	//--- delete and shift 
		IF udiNbOfCarrier >= 1 THEN
			//--- Check if Carrier is outside
				//--- zero is not inside start and end pos 
			FOR udiTraceArrayIndex := 1 TO c_udiTraceObjects DO
				IF audiTraceCarrierIndex[udiTraceArrayIndex] = 0 THEN
					CONTINUE;
				END_IF
				IF i_lrStartPos < i_lrEndPos THEN 
					IF fbMulticarrier.raifCarrier[audiTraceCarrierIndex[udiTraceArrayIndex]].ifFeedback.ifFeedbackMotionValues.lrRefTrackPosition > i_lrEndPos
						OR fbMulticarrier.raifCarrier[audiTraceCarrierIndex[udiTraceArrayIndex]].ifFeedback.ifFeedbackMotionValues.lrRefTrackPosition < i_lrStartPos
					THEN
						xCarrierIsOutside := TRUE;
						EXIT;
					END_IF
					
				//--- zero is inside start and end pos  
				ELSIF i_lrStartPos > i_lrEndPos THEN 
					IF fbMulticarrier.raifCarrier[audiTraceCarrierIndex[udiTraceArrayIndex]].ifFeedback.ifFeedbackMotionValues.lrRefTrackPosition > i_lrEndPos
						AND fbMulticarrier.raifCarrier[audiTraceCarrierIndex[udiTraceArrayIndex]].ifFeedback.ifFeedbackMotionValues.lrRefTrackPosition < i_lrStartPos
					THEN
						xCarrierIsOutside := TRUE;
						EXIT;
					END_IF
				END_IF
			END_FOR
			
			IF xCarrierIsOutside THEN
				xCarrierIsOutside := FALSE;
				udiNbOfCarrier := udiNbOfCarrier -1;
				axCarrierArrayIsBlocked[udiTraceArrayIndex] := FALSE;
				audiTraceCarrierIndex[udiTraceArrayIndex] := 0;
			END_IF
		END_IF
END_METHOD

ACTION ExceptionControl_Action:
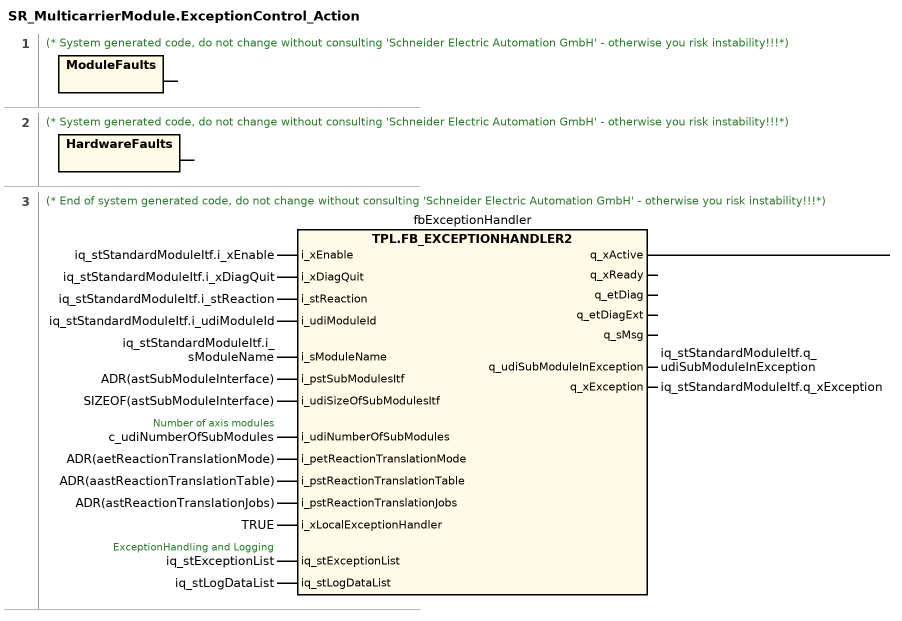
// NETWORK 1
// (* System generated code, do not change without consulting 'Schneider Electric Automation GmbH' - otherwise you risk instability!!!*)
ModuleFaults();

// NETWORK 2
// (* System generated code, do not change without consulting 'Schneider Electric Automation GmbH' - otherwise you risk instability!!!*)
HardwareFaults();

// NETWORK 3
// (* End of system generated code, do not change without consulting 'Schneider Electric Automation GmbH' - otherwise you risk instability!!!*)
//   fbExceptionHandler: ExceptionHandling related variables
//   c_udiNumberOfSubModules: Number of axis modules
//   iq_stExceptionList: ExceptionHandling and Logging
fbExceptionHandler(
    i_xEnable := iq_stStandardModuleItf.i_xEnable,
    i_xDiagQuit := iq_stStandardModuleItf.i_xDiagQuit,
    i_stReaction := iq_stStandardModuleItf.i_stReaction,
    i_udiModuleId := iq_stStandardModuleItf.i_udiModuleId,
    i_sModuleName := iq_stStandardModuleItf.i_sModuleName,
    i_pstSubModulesItf := ADR(astSubModuleInterface),
    i_udiSizeOfSubModulesItf := SIZEOF(astSubModuleInterface),
    i_udiNumberOfSubModules := c_udiNumberOfSubModules,
    i_petReactionTranslationMode := ADR(aetReactionTranslationMode),
    i_pstReactionTranslationTable := ADR(aastReactionTranslationTable),
    i_pstReactionTranslationJobs := ADR(astReactionTranslationJobs),
    i_xLocalExceptionHandler := TRUE,
    iq_stExceptionList := iq_stExceptionList,
    iq_stLogDataList := iq_stLogDataList,
    q_udiSubModuleInException => iq_stStandardModuleItf.q_udiSubModuleInException,
    q_xException => iq_stStandardModuleItf.q_xException); // TPL.FB_EXCEPTIONHANDLER2
END_ACTION

ACTION HardwareFaults:
(* System generated code, do not change without consulting 'Schneider Electric Automation GmbH' - otherwise you risk instability!!! *)
// 
IF SystemConfiguration.G_ifController <> 0 THEN
	diDiagCode := SystemConfiguration.G_ifController.DiagCode; 
	IF diDiagCode <> diDiagCode_old THEN
		diDiagCode_old	:= diDiagCode;
		stDiagSource	:= SystemConfiguration.G_ifController.DiagSource;
		IF 			stDiagSource.udiType = SystemInterface.LXMMCS_TYPE.udiType 
			OR_ELSE stDiagSource.udiType =  SystemInterface.LXMMCC_TYPE.udiType 
		THEN 
			diDiagClass		:= SystemConfiguration.G_ifController.DiagClass;
			sDiagMsg		:= SystemConfiguration.G_ifController.DiagMsg;
			sInstanceName	:= 'UnknownDevice';
			SystemInterface.FC_GetObjNameByLogAddr(i_stLogAdr := stDiagSource, i_diMaxSize := SIZEOF(sInstanceName), iq_sName := sInstanceName);
			sDiagMsgExt := '';
			xSuccess := __QUERYINTERFACE(SystemConfiguration.G_ifController, ifDiagnosis);
			IF xSuccess AND (ifDiagnosis <> 0) THEN
				sDiagMsgExt := ifDiagnosis.DiagExtMsg;
			END_IF

			diDiagClass := SystemConfiguration.G_ifController.DiagClass;
			IF diDiagClass = 4 THEN
				stHardwareException.stReaction.axReaction[TPL.ET_Reaction.AsyncStop]  := TRUE;
				stHardwareException.stReaction.axReaction[TPL.ET_Reaction.SyncStopEL] := FALSE;
				stHardwareException.stReaction.axReaction[TPL.ET_Reaction.SyncStopEH] := FALSE;
			ELSIF diDiagClass = 3 THEN
				stHardwareException.stReaction.axReaction[TPL.ET_Reaction.AsyncStop]  := FALSE;
				stHardwareException.stReaction.axReaction[TPL.ET_Reaction.SyncStopEL] := TRUE;
				stHardwareException.stReaction.axReaction[TPL.ET_Reaction.SyncStopEH] := FALSE;
			ELSIF (diDiagClass = 2 OR diDiagClass = 1) THEN
				stHardwareException.stReaction.axReaction[TPL.ET_Reaction.AsyncStop]  := FALSE;
				stHardwareException.stReaction.axReaction[TPL.ET_Reaction.SyncStopEL] := FALSE;
				stHardwareException.stReaction.axReaction[TPL.ET_Reaction.SyncStopEH] := TRUE;
			END_IF
			
			stHardwareException.etDiag		:= GD.ET_Diag.DiagActive;
			stHardwareException.udiDiagExt	:= ET_DiagExt.SystemFatalException;								
			stHardwareException.sDiagExt	:= FC_EtDiagExtToString(stHardwareException.udiDiagExt);	
			stHardwareException.sMsg		:= PDL.FC_MultiConcat(	i_sString1 := STANDARD.CONCAT(sInstanceName, ' '),
																	i_sString2 := STANDARD.CONCAT(DINT_TO_STRING(diDiagCode), ' '), 
																	i_sString3 := STANDARD.CONCAT(sDiagMsg, ' '), 
																	i_sString4 := sDiagMsgExt);
																	
			stHardwareException.udiExceptionNumber := TPL.FC_GenerateExceptionNumber( i_etSource := TPL.ET_ExceptionSource.System, i_udiDiagExt := DINT_TO_UDINT(diDiagCode) );
			fbExceptionHandler.SetException(i_xExceptionActive	:= TRUE,
											iq_stException		:= stHardwareException,
											iq_stExceptionList	:= iq_stExceptionList);
		END_IF
	END_IF
END_IF
// (* End of system generated code, do not change without consulting 'Schneider Electric Automation GmbH' - otherwise you risk instability!!! *)
END_ACTION

ACTION Init_Exceptions:
(* System generated code, could be modified for your application *)
stUpdateStructsException.etDiag												:= GD.ET_Diag.UnexpectedProgramBehavior;
stUpdateStructsException.udiDiagExt											:= ET_DiagExt.UpdateStructsException;
stUpdateStructsException.sDiagExt											:= FC_EtDiagExtToString(stUpdateStructsException.udiDiagExt);
stUpdateStructsException.sMsg												:= '';	(* Replaced on usage *)
stUpdateStructsException.udiModuleId										:= iq_stStandardModuleItf.i_udiModuleId;
stUpdateStructsException.sModuleName										:= iq_stStandardModuleItf.i_sModuleName;
stUpdateStructsException.stReaction.axReaction[TPL.ET_Reaction.AsyncStop]	:= TRUE;
stUpdateStructsException.etSource											:= TPL.ET_ExceptionSource.NodeModule;
stUpdateStructsException.timDelayTime										:= T#0MS;
stUpdateStructsException.wHmiAttributes										:= 0;
stUpdateStructsException.xAutoQuit											:= FALSE;

stInitReactionsException.etDiag												:= GD.ET_Diag.UnexpectedProgramBehavior;
stInitReactionsException.udiDiagExt											:= ET_DiagExt.InitReactionsException;
stInitReactionsException.sDiagExt											:= FC_EtDiagExtToString(stInitReactionsException.udiDiagExt);
stInitReactionsException.sMsg												:= '';	(* Replaced on usage *)
stInitReactionsException.udiModuleId										:= iq_stStandardModuleItf.i_udiModuleId;
stInitReactionsException.sModuleName										:= iq_stStandardModuleItf.i_sModuleName;
stInitReactionsException.stReaction.axReaction[TPL.ET_Reaction.AsyncStop]	:= TRUE;
stInitReactionsException.etSource											:= TPL.ET_ExceptionSource.NodeModule;
stInitReactionsException.timDelayTime										:= T#0MS;
stInitReactionsException.wHmiAttributes										:= 0;
stInitReactionsException.xAutoQuit											:= FALSE;

stInitSubModulesException.etDiag											:= GD.ET_Diag.UnexpectedProgramBehavior;
stInitSubModulesException.udiDiagExt										:= ET_DiagExt.InitSubModulesException;
stInitSubModulesException.sDiagExt											:= FC_EtDiagExtToString(stInitSubModulesException.udiDiagExt);
stInitSubModulesException.sMsg												:= '';	(* Replaced on usage *)
stInitSubModulesException.udiModuleId										:= iq_stStandardModuleItf.i_udiModuleId;
stInitSubModulesException.sModuleName										:= iq_stStandardModuleItf.i_sModuleName;
stInitSubModulesException.stReaction.axReaction[TPL.ET_Reaction.AsyncStop]	:= TRUE;
stInitSubModulesException.etSource											:= TPL.ET_ExceptionSource.NodeModule;
stInitSubModulesException.timDelayTime										:= T#0MS;
stInitSubModulesException.wHmiAttributes									:= 0;
stInitSubModulesException.xAutoQuit											:= FALSE;

(*------------------------------------------------------------------------------------------*)
(* Init User Exceptions *)

	// TPL.ET_Reaction.AsyncStop
	// TPL.ET_Reaction.SyncStopEL
	// TPL.ET_Reaction.SyncStopEH
	// TPL.ET_Reaction.StopEndOfCycle
	// TPL.ET_Reaction.MainsContactorOff
	
(*------------------------------------------------------------------------------------------*)

stException.etDiag												:= GD.ET_Diag.ExecutionAborted;
stException.udiModuleId											:= iq_stStandardModuleItf.i_udiModuleId;
stException.sModuleName											:= iq_stStandardModuleItf.i_sModuleName;
stException.stReaction.axReaction[TPL.ET_Reaction.SyncStopEH]	:= TRUE;
stException.etSource											:= TPL.ET_ExceptionSource.User;
stException.timDelayTime										:= T#0MS;
stException.wHmiAttributes										:= 0;
stException.xAutoQuit											:= FALSE;

stHardwareException.udiModuleId											:= iq_stStandardModuleItf.i_udiModuleId;
stHardwareException.sModuleName											:= iq_stStandardModuleItf.i_sModuleName;
stHardwareException.udiDiagExt											:= ET_DiagExt.HardwareException ;
stHardwareException.etSource											:= TPL.ET_ExceptionSource.System;
stHardwareException.timDelayTime										:= T#0MS;
stHardwareException.wHmiAttributes										:= 0;
stHardwareException.xAutoQuit											:= FALSE;
END_ACTION

ACTION Init_Reactions:
(* System generated code, only to be changed by experienced programmers *)
IF c_udiNumberOfSubModules < 1 THEN
	RETURN;
END_IF

(* Change of default reactions only on demand *)
(* Compare SR MainMachine Action Init_Reactions *)

xInitReactionsException := FALSE;

(*****************************************************************************************************************************************************)
(* Init ReactionTranslationMode *)

TPL.FC_InitReactionTranslationMode(	i_udiNumberOfSubModules			:= c_udiNumberOfSubModules,
									i_petReactionTranslationMode	:= ADR(aetReactionTranslationMode),
									q_etDiag						=> etDiag,
									q_etDiagExt						=> etDiagExtTPL);
							
IF etDiag <> GD.ET_Diag.Ok AND NOT xInitReactionsException THEN
	xInitReactionsException := TRUE;
	
	stInitReactionsException.sMsg := PDL.FC_MultiConcat(i_sString1 := 'InitReactionTranslationMode - ', 
														i_sString2 := GD.FC_EtDiagToString(i_etDiag := etDiag), 
														i_sString3 := ' - ', 
														i_sString4 := TPL.FC_EtDiagExtToString(i_etDiagExt := etDiagExtTPL));
END_IF	

(*****************************************************************************************************************************************************)
(* Init ReactionTranslationTable *)	

TPL.FC_InitReactionTranslationTable(i_udiNumberOfSubModules			:= c_udiNumberOfSubModules,
									i_pstReactionTranslationTable	:= ADR(aastReactionTranslationTable),
									q_etDiag						=> etDiag,
									q_etDiagExt						=> etDiagExtTPL);
									
IF etDiag <> GD.ET_Diag.Ok AND NOT xInitReactionsException THEN
	xInitReactionsException := TRUE;
	
	stInitReactionsException.sMsg := PDL.FC_MultiConcat(i_sString1 := 'InitReactionTranslationTable - ', 
														i_sString2 := GD.FC_EtDiagToString(i_etDiag := etDiag), 
														i_sString3 := ' - ', 
														i_sString4 := TPL.FC_EtDiagExtToString(i_etDiagExt := etDiagExtTPL));
END_IF		

(*****************************************************************************************************************************************************)
(* Init ReactionTranslationJobs *)	
								
TPL.FC_InitReactionTranslationJobs( i_udiNumberOfSubModules			:= c_udiNumberOfSubModules,
									i_pstReactionTranslationJobs	:= ADR(astReactionTranslationJobs),
									q_etDiag						=> etDiag,
									q_etDiagExt						=> etDiagExtTPL);
						
IF etDiag <> GD.ET_Diag.Ok AND NOT xInitReactionsException THEN
	xInitReactionsException := TRUE;
	
	stInitReactionsException.sMsg := PDL.FC_MultiConcat(i_sString1 := 'InitReactionTranslationJobs - ', 
														i_sString2 := GD.FC_EtDiagToString(i_etDiag := etDiag), 
														i_sString3 := ' - ', 
														i_sString4 := TPL.FC_EtDiagExtToString(i_etDiagExt := etDiagExtTPL));
END_IF		

(*****************************************************************************************************************************************************)
(* Set exception if any exception occurred *)

fbExceptionHandler.SetException(i_xExceptionActive	:= xInitReactionsException, 
								iq_stException		:= stInitReactionsException, 
								iq_stExceptionList	:= iq_stExceptionList);
					
xInitSuccessful := xInitSuccessful AND NOT xInitReactionsException;

etDiag := GD.ET_Diag.Ok;
(* End of system generated code, only to be changed by experienced programmers *)
END_ACTION

ACTION ModuleFaults:
(* System generated code, could be modified for your application *)

//--- Errors Initialization or using MCR/MCRS-library functions in programm
IF xSetException AND NOT xErrorStored THEN
			
	xErrorStored := TRUE;
		
	IF etResultMCRS <> MCRS.ET_Result.Ok THEN
		stException.sDiagExt := TO_STRING(etResultMCRS);
	
	ELSIF etResultMCR <> MCR.ET_Result.Ok THEN
		stException.sDiagExt := TO_STRING(etResultMCR);
	END_IF
			
	stException.sMsg := sResultMsgMCR;
	//--- set Exception  ------------------------------------------------------------									
	fbExceptionHandler.SetException(i_xExceptionActive	:= xSetException,
									iq_stException		:= stException,
									iq_stExceptionList	:= iq_stExceptionList);	
END_IF

ErrorsFromStations();

//--- FB_Multicarrier ------------------------------------------------------------									
IF astSubModuleInterface[c_udiMultiCarrierTrack].q_xException THEN
	stException.udiDiagExt		:= etResultFbMulticarrier;
	stException.sDiagExt		:= TO_STRING(etResultFbMulticarrier);
	stException.sMsg			:= concat('FB_Multicarrier: ',sResultMsgFbMulticarrier);
	xSetException				:= TRUE;
	//--- set Exception  ------------------------------------------------------------									
	fbExceptionHandler.SetException(i_xExceptionActive	:= xSetException,
									iq_stException		:= stException,
									iq_stExceptionList	:= iq_stExceptionList);	
END_IF

//--- FB_CrashPrevention ------------------------------------------------------------									
IF xErrorFbCrashPrevention THEN
	stException.udiDiagExt		:= etResultFbCrashPrevention;
	stException.sDiagExt		:= TO_STRING(etResultFbCrashPrevention);
	stException.sMsg			:= concat('FB_CrashPrevention: ',sResultMsgFbCrashPrevention);
	xSetException				:= TRUE;
	AddMessageToAPL(stException.sMsg);
	//--- set Exception  ------------------------------------------------------------									
	fbExceptionHandler.SetException(i_xExceptionActive	:= xSetException,
									iq_stException		:= stException,
									iq_stExceptionList	:= iq_stExceptionList);	
END_IF

//--- FB_TrackCalibration ------------------------------------------------------------									
IF xErrorFbTrackCalibration THEN
	stException.udiDiagExt		:= etResultFbTrackCalibration;
	stException.sDiagExt		:= TO_STRING(etResultFbTrackCalibration);
	stException.sMsg			:= concat('FB_TrackCalibration: ',sResultMsgFbTrackCalibration);
	xSetException				:= TRUE;
	AddMessageToAPL(stException.sMsg);
	//--- set Exception  ------------------------------------------------------------									
	fbExceptionHandler.SetException(i_xExceptionActive	:= xSetException,
									iq_stException		:= stException,
									iq_stExceptionList	:= iq_stExceptionList);	
END_IF

//--- Auto Mode  ------------------------------------------------------------									
IF NOT xHomingWasSuccessful AND (iq_stStandardModuleItf.q_diCMDActive = ET_Cmd.Auto) AND iq_stStandardModuleItf.q_xCMDActive THEN
	stException.udiDiagExt		:= ET_DiagExt.UnexpectedFeedback;
	stException.sDiagExt		:= FC_EtDiagExtToString(ET_DiagExt.UnexpectedFeedback);
	stException.sMsg			:= 'Auto Mode: Multicarrier not homed';
	xSetException				:= TRUE;
	//--- set Exception  ------------------------------------------------------------									
	fbExceptionHandler.SetException(i_xExceptionActive	:= xSetException,
									iq_stException		:= stException,
									iq_stExceptionList	:= iq_stExceptionList);	
END_IF

//--- ControlEnable  ------------------------------------------------------------									
IF fbTonTimeOutControlEnable.Q THEN
	xCheckTimeOutControlEnable	:= FALSE;
	stException.udiDiagExt		:= ET_DiagExt.TimeoutControlEnable;
	stException.sDiagExt		:= FC_EtDiagExtToString(ET_DiagExt.TimeoutControlEnable);
	stException.sMsg			:= 'ControlEnable: Timeout during Enable/Disable Track';
	xSetException				:= TRUE;
	AddMessageToAPL(stException.sMsg);
	//--- set Exception  ------------------------------------------------------------									
	fbExceptionHandler.SetException(i_xExceptionActive	:= xSetException,
									iq_stException		:= stException,
									iq_stExceptionList	:= iq_stExceptionList);	
END_IF

//--- SegmentNotEnabled  ------------------------------------------------------------									
IF xEnableTrackSuccessful THEN
	FOR udiIndex := 1 TO ifMulticarrier.ifFeedback.ifFeedbackConfiguration.udiNumberOfSegments DO
		IF iq_stMulticarrierModule.i_aifSegmentEnable[udiIndex].State <> 3 THEN
			stException.udiDiagExt		:= ET_DiagExt.SegmentNotEnabled;
			stException.sDiagExt		:= FC_EtDiagExtToString(ET_DiagExt.SegmentNotEnabled);
			stException.sMsg			:= PDL.FC_MultiConcat(	i_sString1 := 'Segment[', 
																i_sString2 := TO_STRING(udiIndex), 
																i_sString3 := '] is not enabled', 
																i_sString4 := '');
			xSetException				:= TRUE;
			AddMessageToAPL(stException.sMsg);
			//--- set Exception  ------------------------------------------------------------									
			fbExceptionHandler.SetException(i_xExceptionActive	:= xSetException,
											iq_stException		:= stException,
											iq_stExceptionList	:= iq_stExceptionList);
			EXIT;
		END_IF
	END_FOR
END_IF

//--- write exception msg in VIS_Multicarrier -> Error	-------------------------------------								
IF xSetException THEN
	sEtResult := stException.sDiagExt;
	FC_SplitString(i_sString:= stException.sMsg, q_sString1=> sResultMsg1, q_sString2=> sResultMsg2, q_sString3=> sResultMsg3);
END_IF

//--- select Error Tab in Vis -------------------------------------									
fbErrorVisTabTrig(CLK := xSetException);
IF fbErrorVisTabTrig.Q THEN
	uiAdditionalVisTabs := 3;
END_IF

//--- select Pos Tab in Vis -------------------------------------									
fbResetErrorVisTabTrig(CLK := xSetException);
IF fbResetErrorVisTabTrig.Q THEN
	uiAdditionalVisTabs := 0;
END_IF

(* end of System generated code, could be modified for your application *)
END_ACTION

ACTION StopAllCarriers:
FOR udiLoop := 1 TO ifMulticarrier.ifFeedback.ifFeedbackConfiguration.udiNumberOfCarriers DO
				
						ifMulticarrier.raifCarrier[udiLoop].ifMotion.StopCarrier(
														q_xError		=> xSetException,
														q_etResult		=> etResultMCR,
														q_sResultMsg	=> sResultMsgMCR);
													
					
				IF xSetException THEN
					sResultMsgMCR := concat('StopCarrier: ',sResultMsgMCR);
					EXIT;
				END_IF
				
			END_FOR
END_ACTION

ACTION ExitLastOpMode:
//-- Auto ---
		IF etLastCmd = ET_Cmd.Auto THEN
			;
			
	//-- Prepare ---
		ELSIF  etLastCmd = ET_Cmd.Prepare THEN
			;
			
	//-- TestMulticarrier ---
// 		ELSIF  etLastCmd = ET_Cmd.TestMulticarrier AND etLastCmd <> iq_stStandardModuleItf.q_diCMDActive THEN
		ELSIF  		etLastCmd = ET_Cmd.TestMulticarrier 
				AND (iq_stStandardModuleItf.q_diCMDActive = ET_Cmd.Prepare OR iq_stStandardModuleItf.q_diCMDActive = ET_Cmd.Auto) 
		THEN
					
				SR_CallTestStations.DeactivateLastTestStation();
				
	//-- TrackCalibration ---
		ELSIF  etLastCmd = ET_Cmd.TrackCalibration THEN
			;
			
	//-- Manual ---
		ELSIF  etLastCmd = ET_Cmd.Manual THEN
			
			Manual_Exit();
			
	//-- Stop ---
		ELSIF  etLastCmd = ET_Cmd.Stop THEN
			;
			
	//-- Abort ---
		ELSIF  etLastCmd = ET_Cmd.Abort THEN
			;
		END_IF
END_ACTION

ACTION MoveAllCarriersInFirstStation:
//--- 1. get carrier with lowest distances to targetposition -----------------
	MCR.FC_OrderOfCarriersToTargetPosition(
			i_xInForwardDirection	:= TRUE, 
			i_lrTargetPosition		:= stStation1.lrWaitStationPosition, 
			i_ifMulticarrier		:= fbMulticarrier, 
			q_udiNumberOfCarriersFound	=> udiNumberOfCarrier,
			q_audiOrderOfCarriers		=> audiOrderOfCarrier,
			q_xError					=> xSetException,
			q_etResult					=> etResultMCR,
			q_sResultMsg				=> sResultMsgMCR);	
			
//
//--- 2. Delete all Product from configuration -------
	IF NOT xSetException THEN
		FOR udiLoop := 1 TO udiNumberOfCarrier  DO
			ifMulticarrier.raifCarrier[udiLoop].ifConfiguration.xProductPresent := FALSE;	
		END_FOR	
	END_IF	
//

//--- 3. Set the minimum gap the Carriers should consider during movement -------
SetMinGapForMoveGapControl();

//--- 4. Send Carriers with MoveGapControl to first station -----------------
	IF NOT xSetException THEN
		FOR udiLoop := 1 TO udiNumberOfCarrier DO
				
			IF NOT xSetException THEN
				ifMulticarrier.raifCarrier[audiOrderOfCarrier[udiLoop]].ifMotion.SetMotionParameter(
						i_lrMaxVelocity		:= stStation1.lrMaxVelocity, 
						i_lrMaxAcceleration	:= stStation1.lrMaxAcceleration, 
						i_lrMaxDeceleration	:= stStation1.lrMaxDeceleration,
						i_lrMaxAbsJerk		:= stStation1.lrMaxJerk,
						q_xError			=> xSetException,
						q_etResult			=> etResultMCR,
						q_sResultMsg		=> sResultMsgMCR);	
			END_IF
				
			IF NOT xSetException THEN
				ifMulticarrier.raifCarrier[audiOrderOfCarrier[udiLoop]].ifMotion.ifMoveGapControl.Start(	
										i_etPosMode 	:= MCR.ET_PosMode.AbsoluteForward,
										i_lrTarget		:= stStation1.lrWaitStationPosition,
										i_lrTargetGap	:= stStation1.lrQueueGapAtWaitPos,
										q_xError		=> xSetException,
										q_etResult		=> etResultMCR,
										q_sResultMsg	=> sResultMsgMCR);	
			END_IF
			
		//--- 5. Add Carriers in the right order to first station
			IF NOT xSetException THEN
				fbStation1.AddCarrier(i_ifCarrier := ifMulticarrier.raifCarrier[audiOrderOfCarrier[udiLoop]],
											q_xError		=> xSetException,
											q_etResult		=> etResultMCRS,
											q_sResultMsg	=> sResultMsgMCR);	
				
			END_IF
			
			IF xSetException THEN
				EXIT;
			END_IF							
		END_FOR
	END_IF

	IF xSetException THEN
		sResultMsgMCR	:= Standard.CONCAT('MoveAllCarrierInFirstStation: ',sResultMsgMCR);
	END_IF
END_ACTION

ACTION SetMinGapForMoveGapControl:
//--- Set Gap distance for MoveGapcontrol-------
		IF NOT xSetException THEN
			FOR udiLoop := 1 TO udiNumberOfCarrier  DO
				
				ifMulticarrier.raifCarrier[udiLoop].ifMotion.SetRefMinGapToCarrierInFront(
					i_lrRefMinGap		:= lrRefMinGapToCarrierInFront,
					q_xError			=> xSetException,
					q_etResult			=> etResultMCR,
					q_sResultMsg		=> sResultMsgMCR);	
				
				IF NOT xSetException THEN	
					ifMulticarrier.raifCarrier[udiLoop].ifMotion.SetRefMinGapToCarrierBehind(
						i_lrRefMinGap 		:= lrRefMinGapToCarrierBehind,
						q_xError			=> xSetException,
						q_etResult			=> etResultMCR,
						q_sResultMsg		=> sResultMsgMCR);	
				END_IF
				
				IF xSetException THEN
					EXIT;
				END_IF
			END_FOR
		END_IF
END_ACTION

METHOD VirtualSetPosOfAllCarriers : BOOL
VAR
    udiLoopSetPos 		: UDINT;
    iCarrierNr 		 	: INT;
    lrTrackLengthSum 	: LREAL;
	lrStepPos			: LREAL;
	lrTrackLength		: lreal;
	lrCarrierDist		: LREAL;
END_VAR
IF GVL_Project.Gc_xVirtualMulticarrier THEN	
		lrTrackLengthSum := ifMulticarrier.ifFeedback.ifFeedbackConfiguration.lrTrackLength;
		lrCarrierDist := SEL(ifMulticarrier.ifFeedback.ifFeedbackConfiguration.xIsClosedRing,
							(lrTrackLengthSum/TO_LREAL(ifMulticarrier.ifFeedback.ifFeedbackConfiguration.udiNumberOfCarriers+1)),
							(lrTrackLengthSum/TO_LREAL(ifMulticarrier.ifFeedback.ifFeedbackConfiguration.udiNumberOfCarriers)));
	
	FOR udiLoopSetPos := 1 TO ifMulticarrier.ifFeedback.ifFeedbackConfiguration.udiNumberOfCarriers DO
		
		ifMulticarrier.raifCarrier[udiLoopSetPos].ifMotion.InitialSetPosVirtualCarrier(
			i_lrSetposValue 	:= lrCarrierDist * (ifMulticarrier.ifFeedback.ifFeedbackConfiguration.udiNumberOfCarriers + 1 - udiLoopSetPos), 
			q_xError			=> xSetException,
			q_etResult			=> etResultMCR,
			q_sResultMsg		=> sResultMsgMCR);
			
		IF xSetException THEN
			sResultMsgMCR	:= concat('VirtualSetPosOfAllCarriers: ',sResultMsgMCR);
			EXIT;
		END_IF
	END_FOR
		
	IF NOT xSetException THEN	
		VirtualSetPosOfAllCarriers := TRUE;
	END_IF
END_IF
END_METHOD

ACTION Init_Carriers:
IF ifMulticarrier <> 0 THEN
	
	//--- Activate Application logger entry for all Carrier  ------------
	IF NOT xSetException THEN
		FOR udiLoop := 1 TO ifMulticarrier.ifFeedback.ifFeedbackConfiguration.udiNumberOfCarriers DO
			ifMulticarrier.raifCarrier[udiLoop].ifConfiguration.ConfigureApplicationLoggerEntries(
						i_xApplicationLoggerEntriesActive 	:= TRUE,
						q_xError							=> xSetException,
						q_etResult							=> etResultMCR,
						q_sResultMsg						=> sResultMsgMCR);
						
			IF xSetException THEN
				stException.udiDiagExt	:= TO_UDINT(etResultMCR);
				stException.sDiagExt	:= TO_STRING(etResultMCR);
				stException.sMsg		:= sResultMsgMCR;
				
				fbExceptionHandler.SetException(i_xExceptionActive	:= TRUE, 
												iq_stException		:= stException, 
												iq_stExceptionList	:= iq_stExceptionList);
				EXIT;
			END_IF
						
		END_FOR
	END_IF	
	
ELSE
	stException.udiDiagExt	:= ET_DiagExt.InvalidConfiguredParameter;
	stException.sDiagExt	:= 'InvalidConfiguredParameter';
	stException.sMsg		:= 'Init_Carriers: ifMulticarrier = 0';
		
	fbExceptionHandler.SetException(i_xExceptionActive	:= TRUE, 
									iq_stException		:= stException, 
									iq_stExceptionList	:= iq_stExceptionList);
	
END_IF
END_ACTION

ACTION Init_CrashPrevention:
stCrashPreventionParameterLocal.lrCrashDistance		:= GVL_Project.G_lrCrashDistance;				
					
fbCrashPrevention.stParameter						:= stCrashPreventionParameterLocal;

fbCrashPrevention.ifMulticarrier					:= ifMulticarrier;
END_ACTION

ACTION Init_FeedbackForVis:
//-------------------------------------------------------------------------------------------------------------------------------------------
//--- Visualization
//-------------------------------------------------------------------------------------------------------------------------------------------
IF NOT xSetException THEN
	//--- replace dummy feedback with real carrier feedback
	FOR udiVisLoop := 1 TO 150 DO
		
		IF udiVisLoop <= ifMulticarrier.ifFeedback.ifFeedbackConfiguration.udiNumberOfCarriers THEN
			aifVisFeedback[udiVisLoop] := fbMulticarrier.raifCarrier[udiVisLoop].ifFeedback;
		END_IF
			
	END_FOR

	
	//--- calculation the sizing rectangle of background of vis buttons
	IF udiDeltaBottomY = 1000 THEN
	 	udiDeltaBottomY := ((ifMulticarrier.ifFeedback.ifFeedbackConfiguration.udiNumberOfCarriers - 1) / 10) * 40;
	END_IF
END_IF
//
END_ACTION

ACTION Init_Track:
//--- Standard template interface ---------
	astSubModuleInterface[c_udiMultiCarrierTrack].i_sModuleName		:= CONCAT(STR1 := iq_stStandardModuleItf.i_sModuleName, STR2 := ': MultiCarrierTrack');
	astSubModuleInterface[c_udiMultiCarrierTrack].i_xLogEnable		:= 	TRUE;
	astSubModuleInterface[c_udiMultiCarrierTrack].i_wLogDataFilter	:= 	UDINT_TO_WORD(TPL.ET_LogDataFilter.ModuleDefault);
	
	
	astSubModuleInterface[c_udiMultiCarrierTrack].q_xActive			:= TRUE;
	astSubModuleInterface[c_udiMultiCarrierTrack].q_xReady			:= TRUE;
	
	astSubModuleInterface[c_udiMultiCarrierTrack].q_dwModuleType	:= TPL.ET_ModuleType.NodeModule;
//
//--- get interface from FB_Multicarrier
ifMulticarrier	:= fbMulticarrier;	
//
IF ifMulticarrier <> 0 THEN

	AddMessageToAPL('------- SR_MulticarrierModule.Init_Track -------');
	
	//--- ConfigureMulticarrierTrack ------------
		IF NOT xSetException THEN
			ifMulticarrier.ifConfiguration.ConfigureMulticarrierTrack(
					i_ifMulticarrierTrack		:= MC_Track_1,
					q_xError					=> xSetException, 
					q_etResult					=> etResultMCR, 
					q_sResultMsg				=> sResultMsgMCR);
		END_IF
		
	//
	//--- ConfigureMulticarrierCarrierPool ------------
		IF NOT xSetException THEN
			ifMulticarrier.ifConfiguration.ConfigureMulticarrierCarrierPool(
					i_ifMulticarrierCarrierPool	:= MC_CarrierPool,
					q_xError					=> xSetException, 
					q_etResult					=> etResultMCR, 
					q_sResultMsg				=> sResultMsgMCR);
		END_IF
		
	//
	//--- ConfigureArrayOfSegments from devices ------------
		IF NOT xSetException THEN
			ifMulticarrier.ifConfiguration.ConfigureArrayOfMulticarrierSegments(
					i_aifMulticarrierSegments	:= iq_stMulticarrierModule.i_aifMulticarrierSegments, 
					i_udiNumberOfSegments		:= GVL_MulticarrierConfiguration.Gc_astTracks[1].udiNumberOfSegments,
					q_xError					=> xSetException, 
					q_etResult					=> etResultMCR, 
					q_sResultMsg				=> sResultMsgMCR);
		END_IF
	
	//
	//--- ConfigureArrayOfMulticarrierCarrier ------------
		IF NOT xSetException THEN
			ifMulticarrier.ifConfiguration.ConfigureArrayOfMulticarrierCarriers(	
					i_aifMulticarrierCarriers	:= iq_stMulticarrierModule.i_aifMulticarrierCarriers, 
					i_udiNumberOfCarriers		:= GVL_Project.G_udiUsedNumberOfCarriers, 
					q_xError					=> xSetException,
					q_etResult					=> etResultMCR,
					q_sResultMsg				=> sResultMsgMCR);
		
		END_IF
	//
	//--- SetEmergencyParameter ------------
		IF NOT xSetException THEN
			ifMulticarrier.ifConfiguration.SetEmergencyParameter(
					i_lrMaxDeceleration		:= lrMaxDecelerationEmergency, 
					i_lrMaxAbsJerk			:= lrMaxAbsJerkEmergency,
					q_xError				=> xSetException, 
					q_etResult				=> etResultMCR, 
					q_sResultMsg			=> sResultMsgMCR);
		END_IF
		
	//
	//--- ConfigDone ------------
		IF NOT xSetException THEN
			ifMulticarrier.ifConfiguration.ConfigDone(
					q_xError				=> xSetException, 
					q_etResult				=> etResultMCR, 
					q_sResultMsg			=> sResultMsgMCR);
		ELSE
			stException.udiDiagExt	:= TO_UDINT(etResultMCR);
			stException.sDiagExt	:= TO_STRING(etResultMCR);
			stException.sMsg		:= concat('SR_MulticarrierModule.Init_Track: ' ,sResultMsgMCR);
				
			fbExceptionHandler.SetException(i_xExceptionActive	:= TRUE, 
											iq_stException		:= stException, 
											iq_stExceptionList	:= iq_stExceptionList);
		END_IF
	//
		
END_IF
END_ACTION

ACTION InitModule_Action:
(* This step is used for initialisations after being enabled *)
(* System generated code, could be modified for your application *)
IF NOT xSetException THEN
	Init_Exceptions();
	
	xInitSuccessful := TRUE;
	
	iq_stStandardModuleItf.q_xActive		:= TRUE;
	iq_stStandardModuleItf.q_xReady			:= FALSE;
	iq_stStandardModuleItf.q_etDiag			:= GD.ET_Diag.Ok;
	iq_stStandardModuleItf.q_udiDiagExt		:= ET_DiagExt.Initializing;
	iq_stStandardModuleItf.q_sDiagExt		:= FC_EtDiagExtToString(ET_DiagExt.Initializing);
	iq_stStandardModuleItf.q_sMsg			:= '';
	
	Init_Exceptions();
	Init_SubModules();
	Init_CmdTables();
	Init_Reactions();
	UpdateStructs();
	(* End of system generated code, do not change without consulting 'Schneider Electric Automation GmbH' - otherwise you risk instability!!!*)
	
	(* System generated code, could be modified for your application *)
	fbLoggerPoint.etLogLevel := APL.ET_LogLevel.UserAction;
	
	fbModuleController.RegisterLoggerPoint(	i_ifParent	:= fbLoggerPoint,
											i_sName		:= 'ModuleController',
											q_etDiag	=> ,
											q_etDiagExt	=> );
	fbExceptionHandler.RegisterLoggerPoint(	i_ifParent	:= fbLoggerPoint,
											i_sName		:= 'ExceptionHandler',
											q_etDiag	=> ,
											q_etDiagExt	=> );
	
	fbMulticarrier.RegisterLoggerPoint(	i_ifParent	:= fbLoggerPoint,
										i_sName		:= 'Multicarrier',
										q_xError	=> ,
										q_etResult	=> );
										
	fbTrackCalibration.RegisterLoggerPoint(	i_ifParent	:= fbLoggerPoint,
											i_sName		:= 'TrackCalibration',
											q_xError	=> ,
											q_etResult	=> );	

	SR_CallTestStations.RegisterLoggerPoint(i_ifParent := fbLoggerPoint);
	

	Init_RegisterStationsToAPL();
	
	Init_Track();
	Init_Carriers();
	Init_FeedbackForVis();
	Init_CrashPrevention();
	
	xInitSuccessful := xInitSuccessful AND NOT xSetException;
	
END_IF

ExceptionControl_Action();

(* End of system generated code, could be modified for your application *)

(* Application specific code *)
(* ToDo: Add your application specific code here *)
;
(* End of application specific code *)
END_ACTION

ACTION Manual_Entry:
AddMessageToAPL('------- Start Opmode: Manual -------');

//--- Setting for Vis_Control ----
xSetJogSingleCarrier 	:= FALSE;
xSetJogAllCarrier 		:= FALSE;
iAxisSelect 			:= 888;
xJogSingleCarrier 		:= TRUE;
xJogAllCarrier 			:= FALSE;
iJogMode 				:= 0;
xJogForw 				:= FALSE;
xJogBack 				:= FALSE;

//--- deactivate all jogging inputs ------------------------------------------------------
IF NOT xSetException THEN
	FOR udiLoop := 1 TO ifMulticarrier.ifFeedback.ifFeedbackConfiguration.udiNumberOfCarriers DO
	
			ifMulticarrier.raifCarrier[udiLoop].ifMotion.ifJogging.xJogForward  := FALSE;
			ifMulticarrier.raifCarrier[udiLoop].ifMotion.ifJogging.xJogBackward := FALSE;
			ifMulticarrier.raifCarrier[udiLoop].ifMotion.ifJogging.xJogSelect 	:= FALSE;
			
			ifMulticarrier.raifCarrier[udiLoop].ifMotion.ifJogging.Stop(
																	q_xError		=> xSetException,
																	q_etResult		=> etResultMCR,
																	q_sResultMsg	=> sResultMsgMCR);	
			
			IF xSetException THEN
				EXIT;
			END_IF
	END_FOR
END_IF

IF NOT xSetException THEN
	FOR udiLoop := 1 TO ifMulticarrier.ifFeedback.ifFeedbackConfiguration.udiNumberOfCarriers DO	
						
	//--- Activate Jogmode in FB_Multicarrier ------------------------------------------------------
		ifMulticarrier.raifCarrier[udiLoop].ifMotion.ifJogging.Start(
				q_xError		=> xSetException,
				q_etResult		=> etResultMCR,
				q_sResultMsg	=> sResultMsgMCR);	
			
		IF xSetException THEN
			EXIT;
		END_IF
		
	END_FOR
END_IF

//--- store min gap ------------------------------------------------------
IF NOT xSetException THEN
	FOR udiLoop := 1 TO ifMulticarrier.ifFeedback.ifFeedbackConfiguration.udiNumberOfCarriers DO
		
		alrStoredMinGapInFront[udiLoop] := ifMulticarrier.raifCarrier[udiLoop].ifFeedback.lrRefMinGapToCarrierInFront;
		alrStoredMinGapBehind[udiLoop]  := ifMulticarrier.raifCarrier[udiLoop].ifFeedback.lrRefMinGapToCarrierBehind;
			
	END_FOR
END_IF

//--- Set Gap for manual mode ------------------------------------------------------
IF NOT xSetException THEN
	FOR udiLoop := 1 TO ifMulticarrier.ifFeedback.ifFeedbackConfiguration.udiNumberOfCarriers DO
		
		ifMulticarrier.raifCarrier[udiLoop].ifMotion.SetRefMinGapToCarrierInFront(
			i_lrRefMinGap		:= lrJogMinDistanceBetweenCarrier,
			q_xError			=> xSetException,
			q_etResult			=> etResultMCR,
			q_sResultMsg		=> sResultMsgMCR);	
		
		IF NOT xSetException THEN	
			ifMulticarrier.raifCarrier[udiLoop].ifMotion.SetRefMinGapToCarrierBehind(
				i_lrRefMinGap 		:= lrJogMinDistanceBetweenCarrier,
				q_xError			=> xSetException,
				q_etResult			=> etResultMCR,
				q_sResultMsg		=> sResultMsgMCR);	
		END_IF
				
		IF xSetException THEN
			EXIT;
		END_IF
	END_FOR
END_IF

IF xSetException THEN
	sResultMsgMCR	:= concat('Manual_entry: ',sResultMsgMCR);
END_IF
END_ACTION

ACTION Manual_Exit:
//--- Set RefMinGap on stored values ------------------------------------------------------
IF NOT xSetException THEN
	FOR udiLoop := 1 TO ifMulticarrier.ifFeedback.ifFeedbackConfiguration.udiNumberOfCarriers DO
		
		ifMulticarrier.raifCarrier[udiLoop].ifMotion.SetRefMinGapToCarrierInFront(
			i_lrRefMinGap		:= alrStoredMinGapInFront[udiLoop],
			q_xError			=> xSetException,
			q_etResult			=> etResultMCR,
			q_sResultMsg		=> sResultMsgMCR);	
		
		IF NOT xSetException THEN	
			ifMulticarrier.raifCarrier[udiLoop].ifMotion.SetRefMinGapToCarrierBehind(
				i_lrRefMinGap 		:= alrStoredMinGapBehind[udiLoop],
				q_xError			=> xSetException,
				q_etResult			=> etResultMCR,
				q_sResultMsg		=> sResultMsgMCR);	
		END_IF
				
		IF xSetException THEN
			EXIT;
		END_IF
	END_FOR
END_IF
END_ACTION

ACTION Manual_Logic:
//--- Set MotionParamter ------------------------------------------------------
	IF lrJogVelocity <> lrJogVelocityOld  THEN
			lrJogVelocityOld 	:= lrJogVelocity;
		
		AddMessageToAPL('------- Manual: SetMotionParameter ------- ');
		
		IF NOT xSetException THEN
			FOR udiLoop := 1 TO ifMulticarrier.ifFeedback.ifFeedbackConfiguration.udiNumberOfCarriers DO	
								
				ifMulticarrier.raifCarrier[udiLoop].ifMotion.SetMotionParameterJogging(
						i_lrMaxVelocity			:= lrJogVelocity, 
						i_lrMaxAcceleration		:= lrJogVelocity, 
						i_lrMaxDeceleration		:= lrJogVelocity * 10, 
						i_lrMaxAbsJerk			:= lrJogVelocity * 100, 		
						q_xError				=> xSetException,
						q_etResult				=> etResultMCR,
						q_sResultMsg			=> sResultMsgMCR);
				
				IF xSetException THEN
					EXIT;
				END_IF
				
				ifMulticarrier.raifCarrier[udiLoop].ifMotion.ifJogging.Start(
						q_xError		=> xSetException,
						q_etResult		=> etResultMCR,
						q_sResultMsg	=> sResultMsgMCR);	
				
				IF xSetException THEN
					EXIT;
				END_IF
				
			END_FOR
		END_IF
	END_IF
	
//
//--- Set min Gap for manual mode ------------------------------------------------------
	IF lrJogMinDistanceBetweenCarrier <> lrJogMinDistanceBetweenCarrierOld THEN
		lrJogMinDistanceBetweenCarrierOld := lrJogMinDistanceBetweenCarrier;
		
		AddMessageToAPL('------- Manual: SetRefMinGap ------- ');
		
		IF NOT xSetException THEN
			FOR udiLoop := 1 TO ifMulticarrier.ifFeedback.ifFeedbackConfiguration.udiNumberOfCarriers DO
				ifMulticarrier.raifCarrier[udiLoop].ifMotion.SetRefMinGapToCarrierBehind(
						i_lrRefMinGap := lrJogMinDistanceBetweenCarrier,
						q_xError				=> xSetException,
						q_etResult				=> etResultMCR,
						q_sResultMsg			=> sResultMsgMCR);
						
				IF xSetException THEN
					EXIT;
				END_IF
				
				ifMulticarrier.raifCarrier[udiLoop].ifMotion.SetRefMinGapToCarrierInFront(
						i_lrRefMinGap := lrJogMinDistanceBetweenCarrier,
						q_xError				=> xSetException,
						q_etResult				=> etResultMCR,
						q_sResultMsg			=> sResultMsgMCR);
						
				IF xSetException THEN
					EXIT;
				END_IF
			END_FOR
		END_IF
	
	END_IF
//
//--- Select Jog Mode ------------------------------------------------------
	CASE iJogMode OF
		
	0:	IF xSetJogAllCarrier THEN
			xSetJogAllCarrier := FALSE;
			iAxisSelect 	  := 999;
			xJogSingleCarrier := FALSE;
			xJogAllCarrier	  := TRUE;
			iJogMode 		  := 10;
		
		ELSIF xSetJogSingleCarrier THEN
			xSetJogSingleCarrier := FALSE;
			iAxisSelect 		 := 888;
			xJogSingleCarrier 	 := TRUE;
			xJogAllCarrier 		 := FALSE;
			iJogMode 			 := 10;
		END_IF
		
	10:	// Deactivate all JogInputs
		FOR udiLoop := 1 TO ifMulticarrier.ifFeedback.ifFeedbackConfiguration.udiNumberOfCarriers DO	
			ifMulticarrier.raifCarrier[udiLoop].ifMotion.ifJogging.xJogForward  := FALSE;
			ifMulticarrier.raifCarrier[udiLoop].ifMotion.ifJogging.xJogBackward := FALSE;
			ifMulticarrier.raifCarrier[udiLoop].ifMotion.ifJogging.xJogSelect := FALSE;
		END_FOR		
		
		iJogMode := 0;
 	
	END_CASE

//
//--- Jog ALL Carrier	---------------------------------------------------------------------------------	
	IF iAxisSelect = 999 THEN
		
		FOR udiLoop := 1 TO ifMulticarrier.ifFeedback.ifFeedbackConfiguration.udiNumberOfCarriers DO
			
			ifMulticarrier.raifCarrier[udiLoop].ifMotion.ifJogging.xJogSelect := TRUE;
			
			IF 	xJogForw AND NOT xJogBack
			THEN
				ifMulticarrier.raifCarrier[udiLoop].ifMotion.ifJogging.xJogForward  := TRUE;
				ifMulticarrier.raifCarrier[udiLoop].ifMotion.ifJogging.xJogBackward := FALSE;
				
			ELSIF xJogBack AND NOT xJogForw 
			THEN
				ifMulticarrier.raifCarrier[udiLoop].ifMotion.ifJogging.xJogForward  := FALSE;
				ifMulticarrier.raifCarrier[udiLoop].ifMotion.ifJogging.xJogBackward := TRUE;
				
			ELSE
				ifMulticarrier.raifCarrier[udiLoop].ifMotion.ifJogging.xJogForward  := FALSE;
				ifMulticarrier.raifCarrier[udiLoop].ifMotion.ifJogging.xJogBackward := FALSE;
				
			END_IF
			
		END_FOR	
	

//
// Jog Carrier from a selection array	-------------------------------------------------------	
	ELSIF iAxisSelect = 888 THEN
		
		//--- set carrier for jogging from vis
		IF xSetCarrierForJoggingFromVis THEN
			xSetCarrierForJoggingFromVis := FALSE;
			
			IF ifMulticarrier.raifCarrier[udiJoggingCarrierNr].ifMotion.ifJogging.xJogSelect THEN
				ifMulticarrier.raifCarrier[udiJoggingCarrierNr].ifMotion.ifJogging.xJogSelect := FALSE;
			ELSE
				ifMulticarrier.raifCarrier[udiJoggingCarrierNr].ifMotion.ifJogging.xJogSelect := TRUE;
			END_IF
		END_IF
		
		xJogCarrierSelectEnableFlag	:= TRUE;
		
		FOR udiLoop := 1 TO ifMulticarrier.ifFeedback.ifFeedbackConfiguration.udiNumberOfCarriers DO
			
			IF 	xJogForw AND NOT xJogBack
			THEN
				IF ifMulticarrier.raifCarrier[udiLoop].ifMotion.ifJogging.xJogSelect
					AND ifMulticarrier.raifCarrier[udiLoop].ifFeedback.ifFeedbackToInFront.lrGapToCarrierInFront 
						> ifMulticarrier.raifCarrier[udiLoop].ifFeedback.ifFeedbackToInFront.lrRefMinGapToCarrierInFront
				THEN
					ifMulticarrier.raifCarrier[udiLoop].ifMotion.ifJogging.xJogForward  := TRUE;
					ifMulticarrier.raifCarrier[udiLoop].ifMotion.ifJogging.xJogBackward := FALSE;
				ELSE
					ifMulticarrier.raifCarrier[udiLoop].ifMotion.ifJogging.xJogForward  := FALSE;
					ifMulticarrier.raifCarrier[udiLoop].ifMotion.ifJogging.xJogBackward := FALSE;
				END_IF
				
			ELSIF 	xJogBack AND NOT xJogForw
			THEN
				IF ifMulticarrier.raifCarrier[udiLoop].ifMotion.ifJogging.xJogSelect
					AND ifMulticarrier.raifCarrier[udiLoop].ifFeedback.ifFeedbackToBehind.lrGapToCarrierBehind 
						> ifMulticarrier.raifCarrier[udiLoop].ifFeedback.ifFeedbackToBehind.lrRefMinGapToCarrierBehind
				THEN
					ifMulticarrier.raifCarrier[udiLoop].ifMotion.ifJogging.xJogForward  := FALSE;
					ifMulticarrier.raifCarrier[udiLoop].ifMotion.ifJogging.xJogBackward := TRUE;
				ELSE
					ifMulticarrier.raifCarrier[udiLoop].ifMotion.ifJogging.xJogForward  := FALSE;
					ifMulticarrier.raifCarrier[udiLoop].ifMotion.ifJogging.xJogBackward := FALSE;
				END_IF
				
			ELSE
					ifMulticarrier.raifCarrier[udiLoop].ifMotion.ifJogging.xJogForward  := FALSE;
					ifMulticarrier.raifCarrier[udiLoop].ifMotion.ifJogging.xJogBackward := FALSE;
			END_IF
			
		END_FOR	
			
	ELSE
		xJogSingleCarrier := FALSE;
		xJogAllCarrier	  := FALSE;			
	END_IF
	
	
	IF xSetException THEN
		sResultMsgMCR	:= concat('Manual_Logic: ',sResultMsgMCR);
	END_IF
END_ACTION

METHOD RegisterLoggerPoint
VAR_INPUT
	i_ifParent	: APL.IF_LoggerPoint;
	i_sName		: STRING[80];
END_VAR
VAR_OUTPUT
	q_etDiag	: GD.ET_Diag := GD.ET_Diag.Ok;
	q_etDiagExt	: ET_DiagExt := ET_DiagExt.Ok;
END_VAR
fbLoggerPoint.RegisterLoggerPoint(	i_ifParent	:= i_ifParent,
									i_sName		:= i_sName,
									i_sType		:= 'Node Module',
									i_sSource	:= 'Program',
									q_etDiag	=> ,
									q_etDiagExt	=> );
END_METHOD

ACTION CallAllStations:
SetStationTriggerViaTimer();

ParameterStation1();

TraceStations();

fbStation1.CyclicMotionCall(iq_xTrigger := stStation1.xTrigger);
END_ACTION

ACTION DeleteAllCarriersFromStations:
fbStation1.CleanUp();
END_ACTION

ACTION ErrorQuitStations:
fbStation1.xErrorQuit 		:= TRUE;
END_ACTION

ACTION ErrorsFromStations:
//--- Errors from station1
IF fbStation1.xError THEN
	xSetException 					:= fbStation1.xError;
	stException.sMsg 				:= fbStation1.sResultMsg;
	stException.sDiagExt 			:= fbStation1.sEtResult;
	stException.udiDiagExt 			:= fbStation1.udiEtResult;
	stException.udiModuleId			:= iq_stStandardModuleItf.i_udiModuleId * 100 +  fbStation1.udiStationId; 
	stException.udiExceptionNumber 	:= TO_UDINT(fbStation1.etResultSource) * 10000 + stException.udiDiagExt;
	//--- set Exception  ------------------------------------------------------------									
	fbExceptionHandler.SetException(i_xExceptionActive	:= xSetException,
									iq_stException		:= stException,
									iq_stExceptionList	:= iq_stExceptionList);	
END_IF
END_ACTION

ACTION Init_RegisterStationsToAPL:
//-- Register Station1 ---------------
IF NOT xSetException THEN
	fbStation1.sName := 'Station1';
	fbStation1.RegisterLoggerPoint(i_ifParent 	  := fbLoggerPoint,
									q_xError	  => xSetException, 
									q_etResult	  => etResultMCRS, 
									q_sResultMsg  => sResultMsgMCR);
END_IF

//-- Register Station2 ---------------
//-- Register Station3 ---------------
// ...
//-- Register Station-n



//-- Report Error -----------------------------------------------------------------
IF xSetException THEN
	stException.udiDiagExt	:= TO_UDINT(etResultMCRS);
	stException.sDiagExt	:= TO_STRING(etResultMCRS);
	stException.sMsg		:= concat('Init_RegisterStationsToAPL: ' ,sResultMsgMCR);

	fbExceptionHandler.SetException(i_xExceptionActive	:= TRUE, 
									iq_stException		:= stException, 
									iq_stExceptionList	:= iq_stExceptionList);
END_IF
END_ACTION

ACTION ParameterStation1:
IF NOT stStation1.xInitParameter THEN
 	stStation1.xInitParameter	:= TRUE;
	
	stStation1.ifTargetStation			:= fbStation1;
	
	stStation1.udiStationId				:= 1;

	stStation1.lrMaxVelocity			:= 850;  
	stStation1.lrMaxAcceleration        := 8500; 
	stStation1.lrMaxDeceleration        := 8500; 
	stStation1.lrMaxJerk                := 85000;
	
	stStation1.lrProcessPos             := 1000;          
	stStation1.lrProcessGap			    := 50; 
	stStation1.lrWaitStationPosition    := 600;   
	stStation1.lrQueueGapAtWaitPos      := 10;  
	
	stStation1.diWaitingTime			:= 100; //= 100ms
END_IF
	
//--- Station1 -------------------------------------------------------
fbStation1.SetStationParameter(
		i_udiStationId			:= stStation1.udiStationId,
		i_ifTargetStation		:= stStation1.ifTargetStation,
		i_lrProcessPosition 	:= stStation1.lrProcessPos,
		i_lrProcessGap			:= stStation1.lrProcessGap,
		i_lrWaitPosition		:= stStation1.lrWaitStationPosition,		
		i_lrWaitGap				:= stStation1.lrQueueGapAtWaitPos,
		i_etStationType			:= ET_StationType.Load,
		i_lrMaxVelocity			:= stStation1.lrMaxVelocity,
		i_lrMaxAcceleration		:= stStation1.lrMaxAcceleration,
		i_lrMaxDeceleration		:= stStation1.lrMaxDeceleration,
		i_lrMaxJerk				:= stStation1.lrMaxJerk );

		
fbStation1.xActivateAPLEntriesForMovedCarriers  	:= stStation1.xApplicationLoggerEntriesActive;
fbStation1.xEnableActivationOfAPLEntriesForCarriers	:= GVL_Project.G_xEnableAplEntriesViaStation;

                                                  	
//--- Emulation ----------------------------------------------------------------------------
	//--- Signals for Machine Expert Twin --- 
		// --- Stations
		GVL_Project.G_astEmulationStations[stStation1.udiStationId].sTextLabel			:= 'Station1';
		GVL_Project.G_astEmulationStations[stStation1.udiStationId].lrWaitPosition 		:= stStation1.lrWaitStationPosition;
		GVL_Project.G_astEmulationStations[stStation1.udiStationId].lrProcessPosition	:= stStation1.lrProcessPos;
		GVL_Project.G_astEmulationStations[stStation1.udiStationId].udiColor			:= DTC.ET_EmulationColors.Black;
		GVL_Project.G_astEmulationStations[stStation1.udiStationId].udiStationId		:= stStation1.udiStationId;
END_ACTION

ACTION ParameterStation2:
IF NOT ststation2.xInitParameter THEN
 	ststation2.xInitParameter	:= TRUE;
	
	ststation2.ifTargetStation			:= fbstation2;
	
	ststation2.udiStationId				:= 2;

	ststation2.lrMaxVelocity			:= 850;  
	ststation2.lrMaxAcceleration        := 8500; 
	ststation2.lrMaxDeceleration        := 8500; 
	ststation2.lrMaxJerk                := 85000;
	
	ststation2.lrProcessPos             := 1000;          
	ststation2.lrProcessGap			    := 50; 
	ststation2.lrWaitStationPosition    := 600;   
	ststation2.lrQueueGapAtWaitPos      := 10;  
	
	ststation2.diWaitingTime			:= 100; //= 100ms
END_IF
	
//--- station2 -------------------------------------------------------
fbstation2.SetStationParameter(
		i_udiStationId			:= ststation2.udiStationId,
		i_ifTargetStation		:= ststation2.ifTargetStation,
		i_lrProcessPosition 	:= ststation2.lrProcessPos,
		i_lrProcessGap			:= ststation2.lrProcessGap,
		i_lrWaitPosition		:= ststation2.lrWaitStationPosition,		
		i_lrWaitGap				:= ststation2.lrQueueGapAtWaitPos,
		i_etStationType			:= ET_StationType.Load,
		i_lrMaxVelocity			:= ststation2.lrMaxVelocity,
		i_lrMaxAcceleration		:= ststation2.lrMaxAcceleration,
		i_lrMaxDeceleration		:= ststation2.lrMaxDeceleration,
		i_lrMaxJerk				:= ststation2.lrMaxJerk );

		
fbstation2.xActivateAPLEntriesForMovedCarriers  	:= ststation2.xApplicationLoggerEntriesActive;
fbstation2.xEnableActivationOfAPLEntriesForCarriers	:= GVL_Project.G_xEnableAplEntriesViaStation;

                                                  	
//--- Emulation ----------------------------------------------------------------------------
	//--- Signals for Machine Expert Twin --- 
		// --- Stations
		GVL_Project.G_astEmulationStations[ststation2.udiStationId].sTextLabel			:= 'station2';
		GVL_Project.G_astEmulationStations[ststation2.udiStationId].lrWaitPosition 		:= ststation2.lrWaitStationPosition;
		GVL_Project.G_astEmulationStations[ststation2.udiStationId].lrProcessPosition	:= ststation2.lrProcessPos;
		GVL_Project.G_astEmulationStations[ststation2.udiStationId].udiColor			:= DTC.ET_EmulationColors.Black;
		GVL_Project.G_astEmulationStations[ststation2.udiStationId].udiStationId		:= ststation2.udiStationId;
END_ACTION

ACTION SetStationTriggerViaTimer:
IF xSetStationTriggerViaTimer THEN
	
	//--- timer Station1
		//--- set timer
		IF 		NOT stStation1.xStartTimer	
			AND fbStation1.xStationReadyForJob 
		THEN
			stStation1.diActualTime := LMC_PacDrive.Timer1;
			stStation1.xStartTimer  := TRUE;
		END_IF
		
		//--- reset timer
		IF 		stStation1.xStartTimer	
			AND LMC_PacDrive.Timer1 > (stStation1.diActualTime + stStation1.diWaitingTime)
		THEN
			stStation1.xTrigger 	 := TRUE;
			stStation1.xStartTimer	 := FALSE;
		END_IF

ELSE
		stStation1.xStartTimer := FALSE;
END_IF
END_ACTION

ACTION TraceStations:
IF etTraceSource = ET_TraceSource.Station1 
		THEN
			SR_CarriersInStationToTrace.Call(
										i_xTrigger := stStation1.xTrigger,
										i_ifStation := fbStation1);
		END_IF
END_ACTION

ACTION StoreCurrentMoveCmds:
//-- Auto ---
		IF etLastCmd = ET_Cmd.Auto THEN
			;
			
	//-- TestMulticarrier ---
		ELSIF  etLastCmd = ET_Cmd.TestMulticarrier THEN
			
			IF SR_CallTestStations.uiSetOpModeTestVis = 2 //= PosAndSync 
			THEN
				SR_PosAndSync.StoreCurrentMoveCmds();
			END_IF
			
		END_IF
END_ACTION

ACTION Input_Action:
(* System generated code, do not change without consulting 'Schneider Electric Automation GmbH' - otherwise you risk instability!!!*)
UpdateStructs();
(* End of system generated code, do not change without consulting 'Schneider Electric Automation GmbH' - otherwise you risk instability!!!*)

xErrorActive := 	iq_stStandardModuleItf.i_stReaction.axReaction[TPL.ET_Reaction.AsyncStop]	
				OR  iq_stStandardModuleItf.i_stReaction.axReaction[TPL.ET_Reaction.SyncStopEL]
				OR  iq_stStandardModuleItf.i_stReaction.axReaction[TPL.ET_Reaction.SyncStopEH]
				OR  iq_stStandardModuleItf.i_stReaction.axReaction[TPL.ET_Reaction.StopEndOfCycle]
				OR  iq_stStandardModuleItf.i_stReaction.axReaction[TPL.ET_Reaction.MainsContactorOff];
END_ACTION

ACTION Logger_Action:
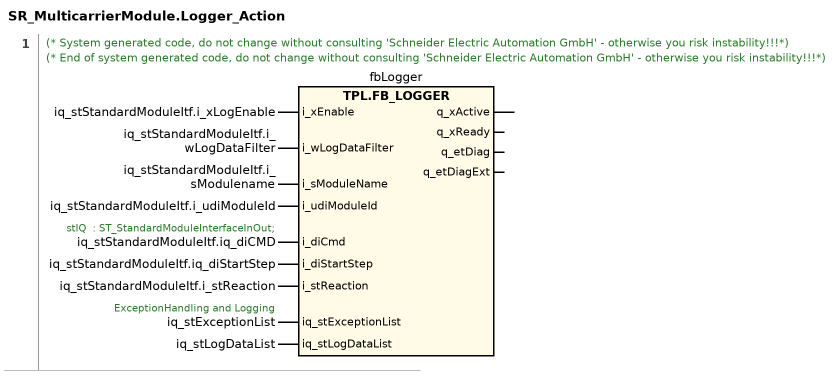
// NETWORK 1
// 					(* System generated code, do not change without consulting 'Schneider Electric Automation GmbH' - otherwise you risk instability!!!*)
// (* End of system generated code, do not change without consulting 'Schneider Electric Automation GmbH' - otherwise you risk instability!!!*)
//
//   fbLogger: Logging related variables
//   iq_stStandardModuleItf.iq_diCMD: stIQ : ST_StandardModuleInterfaceInOut;
//   iq_stExceptionList: ExceptionHandling and Logging
fbLogger(
    i_xEnable := iq_stStandardModuleItf.i_xLogEnable,
    i_wLogDataFilter := iq_stStandardModuleItf.i_wLogDataFilter,
    i_sModuleName := iq_stStandardModuleItf.i_sModulename,
    i_udiModuleId := iq_stStandardModuleItf.i_udiModuleId,
    i_diCmd := iq_stStandardModuleItf.iq_diCMD,
    i_diStartStep := iq_stStandardModuleItf.iq_diStartStep,
    i_stReaction := iq_stStandardModuleItf.i_stReaction,
    iq_stExceptionList := iq_stExceptionList,
    iq_stLogDataList := iq_stLogDataList); // TPL.FB_LOGGER
END_ACTION

ACTION Logic_active:
TraceAndAPL();

//--- Write Crash distance setting from visualization
IF GVL_Project.G_lrCrashDistance <> stCrashPreventionParameterLocal.lrCrashDistance THEN
	stCrashPreventionParameterLocal.lrCrashDistance		:= GVL_Project.G_lrCrashDistance;				
	fbCrashPrevention.stParameter						:= stCrashPreventionParameterLocal;
END_IF
END_ACTION

ACTION Output_Active:
(* System generated code, only to be changed by experienced programmers *)
IF iq_stStandardModuleItf.q_udiSubModuleInException <> 0 THEN
	iq_stStandardModuleItf.q_etDiag		:= GD.ET_Diag.Ok;
	iq_stStandardModuleItf.q_udiDiagExt	:= ET_DiagExt.SubModuleInException;
	iq_stStandardModuleItf.q_sDiagExt		:= FC_EtDiagExtToString(ET_DiagExt.SubModuleInException);
	iq_stStandardModuleItf.q_sMsg			:= '';
ELSE
	IF etDiagModuleController = GD.ET_Diag.Ok THEN
		iq_stStandardModuleItf.q_etDiag	:= etDiagModuleController;
		iq_stStandardModuleItf.q_sMsg		:= sMsgModuleController;
		
		CASE etDiagExtModuleController OF
			TPL.ET_DiagExt.DeactivatingSubModules : 
				iq_stStandardModuleItf.q_udiDiagExt	:= ET_DiagExt.DeactivatingSubModules;
				iq_stStandardModuleItf.q_sDiagExt		:= FC_EtDiagExtToString(ET_DiagExt.DeactivatingSubModules);
			TPL.ET_DiagExt.Disabled : 
				iq_stStandardModuleItf.q_udiDiagExt	:= ET_DiagExt.Disabled;
				iq_stStandardModuleItf.q_sDiagExt		:= FC_EtDiagExtToString(ET_DiagExt.Disabled);
			TPL.ET_DiagExt.ExecuteStep : 
				iq_stStandardModuleItf.q_udiDiagExt	:= ET_DiagExt.ExecuteStep;
				iq_stStandardModuleItf.q_sDiagExt		:= FC_EtDiagExtToString(ET_DiagExt.ExecuteStep);
			TPL.ET_DiagExt.Initializing : 
				iq_stStandardModuleItf.q_udiDiagExt	:= ET_DiagExt.Initializing;
				iq_stStandardModuleItf.q_sDiagExt		:= FC_EtDiagExtToString(ET_DiagExt.Initializing);
			TPL.ET_DiagExt.WaitAtNegativeStep : 
				iq_stStandardModuleItf.q_udiDiagExt	:= ET_DiagExt.WaitAtNegativeStep;
				iq_stStandardModuleItf.q_sDiagExt		:= FC_EtDiagExtToString(ET_DiagExt.WaitAtNegativeStep);
			TPL.ET_DiagExt.WaitCmdsDone : 
				iq_stStandardModuleItf.q_udiDiagExt	:= ET_DiagExt.WaitCmdsDone;
				iq_stStandardModuleItf.q_sDiagExt		:= FC_EtDiagExtToString(ET_DiagExt.WaitCmdsDone);
			TPL.ET_DiagExt.WaitForCmd : 
				iq_stStandardModuleItf.q_udiDiagExt	:= ET_DiagExt.WaitForCmd;
				iq_stStandardModuleItf.q_sDiagExt		:= FC_EtDiagExtToString(ET_DiagExt.WaitForCmd);
			ELSE
				iq_stStandardModuleItf.q_etDiag		:= GD. ET_Diag.UnexpectedProgramBehavior;
				iq_stStandardModuleItf.q_udiDiagExt	:= ET_DiagExt.UnknownStateModuleController;
				iq_stStandardModuleItf.q_sDiagExt		:= FC_EtDiagExtToString(ET_DiagExt.UnknownStateModuleController);
		END_CASE
	ELSE
		iq_stStandardModuleItf.q_etDiag		:= GD.ET_Diag.DiagActive;
		iq_stStandardModuleItf.q_udiDiagExt	:= ET_DiagExt.ModuleControllerException;
		iq_stStandardModuleItf.q_sDiagExt		:= FC_EtDiagExtToString(ET_DiagExt.ModuleControllerException);
		iq_stStandardModuleItf.q_sMsg			:= PDL.FC_MultiConcat(	i_sString1 := GD.FC_EtDiagToString(i_etDiag := etDiagModuleController), 
																			i_sString2 := ' - ',
																			i_sString3 := TPL.FC_EtDiagExtToString(etDiagExtModuleController), 
																			i_sString4 := '');
	END_IF
END_IF

(* End of system generated code, only to be changed by experienced programmers *)
END_ACTION

ACTION Start_Action:
(* This step is active until the machine is being enabled *)

	(* System generated code, do not change without consulting 'Schneider Electric Automation GmbH' - otherwise you risk instability!!! *)
	iq_stStandardModuleItf.q_xActive			:= FALSE;
	iq_stStandardModuleItf.q_xReady				:= FALSE;
	
	iq_stStandardModuleItf.q_etDiag				:= GD.ET_Diag.Ok;
	iq_stStandardModuleItf.q_udiDiagExt			:= ET_DiagExt.Disabled;
	iq_stStandardModuleItf.q_sDiagExt			:= FC_EtDiagExtToString(iq_stStandardModuleItf.q_udiDiagExt);
	iq_stStandardModuleItf.q_sMsg				:= '';
	
	iq_stStandardModuleItf.q_dwModuleType		:= TPL.ET_ModuleType.NodeModule;
	iq_stStandardModuleItf.q_sModuleTypeName	:= 'NodeModule';
	iq_stStandardModuleItf.q_udiModuleVersion	:= 1;	
	(* End of system generated code, do not change without consulting 'Schneider Electric Automation GmbH' - otherwise you risk instability!!! *)
	
	(* System generated code, to be changed by experienced programmers *)
	IF iq_stStandardModuleItf.iq_diCMD <> 0 AND NOT iq_stStandardModuleItf.i_xEnable THEN
		iq_stStandardModuleItf.iq_diCMD := 0;
	END_IF
	(* End of system generated code, to be changed by experienced programmers *)
	

(* Application specific code *)
(* ToDo: Add your application specific code here *)
;
(* End of application specific code *)
END_ACTION

ACTION SubModules_Action:
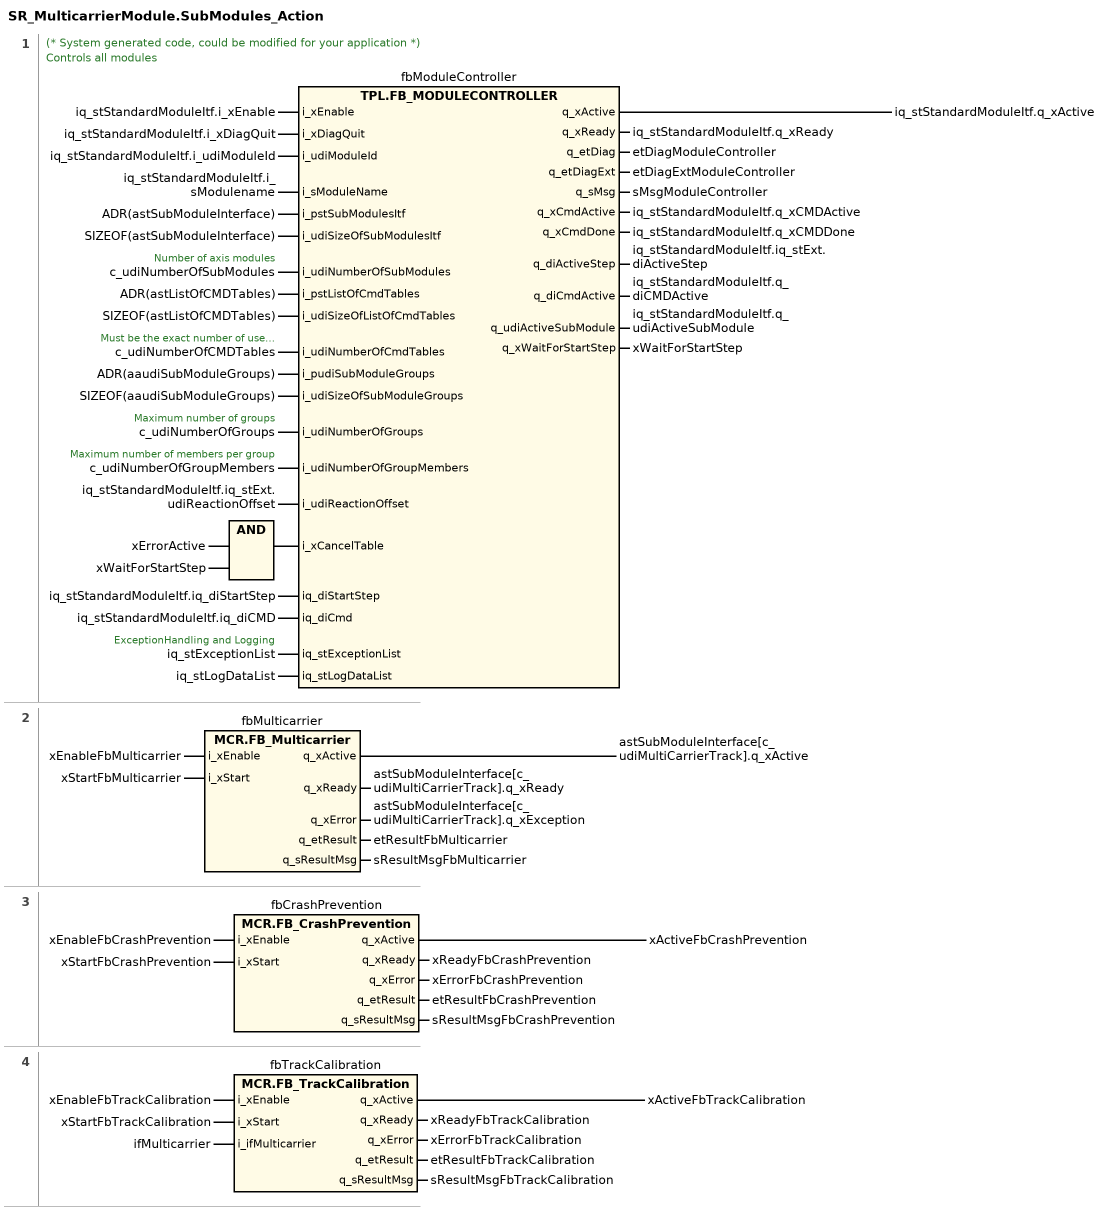
// NETWORK 1
// 					(* System generated code, could be modified for your application *)
// Controls all modules
//
//   fbModuleController: Modules related variables
//   c_udiNumberOfSubModules: Number of axis modules
//   c_udiNumberOfCMDTables: Must be the exact number of used CMDTables!
//   c_udiNumberOfGroups: Maximum number of groups
//   c_udiNumberOfGroupMembers: Maximum number of members per group
//   iq_stExceptionList: ExceptionHandling and Logging
fbModuleController(
    i_xEnable := iq_stStandardModuleItf.i_xEnable,
    i_xDiagQuit := iq_stStandardModuleItf.i_xDiagQuit,
    i_udiModuleId := iq_stStandardModuleItf.i_udiModuleId,
    i_sModuleName := iq_stStandardModuleItf.i_sModulename,
    i_pstSubModulesItf := ADR(astSubModuleInterface),
    i_udiSizeOfSubModulesItf := SIZEOF(astSubModuleInterface),
    i_udiNumberOfSubModules := c_udiNumberOfSubModules,
    i_pstListOfCmdTables := ADR(astListOfCMDTables),
    i_udiSizeOfListOfCmdTables := SIZEOF(astListOfCMDTables),
    i_udiNumberOfCmdTables := c_udiNumberOfCMDTables,
    i_pudiSubModuleGroups := ADR(aaudiSubModuleGroups),
    i_udiSizeOfSubModuleGroups := SIZEOF(aaudiSubModuleGroups),
    i_udiNumberOfGroups := c_udiNumberOfGroups,
    i_udiNumberOfGroupMembers := c_udiNumberOfGroupMembers,
    i_udiReactionOffset := iq_stStandardModuleItf.iq_stExt.udiReactionOffset,
    i_xCancelTable := xErrorActive AND xWaitForStartStep,
    iq_diStartStep := iq_stStandardModuleItf.iq_diStartStep,
    iq_diCmd := iq_stStandardModuleItf.iq_diCMD,
    iq_stExceptionList := iq_stExceptionList,
    iq_stLogDataList := iq_stLogDataList,
    q_xReady => iq_stStandardModuleItf.q_xReady,
    q_etDiag => etDiagModuleController,
    q_etDiagExt => etDiagExtModuleController,
    q_sMsg => sMsgModuleController,
    q_xCmdActive => iq_stStandardModuleItf.q_xCMDActive,
    q_xCmdDone => iq_stStandardModuleItf.q_xCMDDone,
    q_diActiveStep => iq_stStandardModuleItf.iq_stExt.diActiveStep,
    q_diCmdActive => iq_stStandardModuleItf.q_diCMDActive,
    q_udiActiveSubModule => iq_stStandardModuleItf.q_udiActiveSubModule,
    q_xWaitForStartStep => xWaitForStartStep); // TPL.FB_MODULECONTROLLER
iq_stStandardModuleItf.q_xActive := fbModuleController.q_xActive;

// NETWORK 2
fbMulticarrier(
    i_xEnable := xEnableFbMulticarrier,
    i_xStart := xStartFbMulticarrier,
    q_xReady => astSubModuleInterface[c_udiMultiCarrierTrack].q_xReady,
    q_xError => astSubModuleInterface[c_udiMultiCarrierTrack].q_xException,
    q_etResult => etResultFbMulticarrier,
    q_sResultMsg => sResultMsgFbMulticarrier); // MCR.FB_Multicarrier
astSubModuleInterface[c_udiMultiCarrierTrack].q_xActive := fbMulticarrier.q_xActive;

// NETWORK 3
fbCrashPrevention(
    i_xEnable := xEnableFbCrashPrevention,
    i_xStart := xStartFbCrashPrevention,
    q_xReady => xReadyFbCrashPrevention,
    q_xError => xErrorFbCrashPrevention,
    q_etResult => etResultFbCrashPrevention,
    q_sResultMsg => sResultMsgFbCrashPrevention); // MCR.FB_CrashPrevention
xActiveFbCrashPrevention := fbCrashPrevention.q_xActive;

// NETWORK 4
fbTrackCalibration(
    i_xEnable := xEnableFbTrackCalibration,
    i_xStart := xStartFbTrackCalibration,
    i_ifMulticarrier := ifMulticarrier,
    q_xReady => xReadyFbTrackCalibration,
    q_xError => xErrorFbTrackCalibration,
    q_etResult => etResultFbTrackCalibration,
    q_sResultMsg => sResultMsgFbTrackCalibration); // MCR.FB_TrackCalibration
xActiveFbTrackCalibration := fbTrackCalibration.q_xActive;
END_ACTION

ACTION UpdateStructs:
(* System generated code, do not change without consulting 'Schneider Electric Automation GmbH' - otherwise you risk instability!!!*)
fbDetectOnlineChange(	i_xEnable	:= TRUE, 
						i_xDetect	:= TRUE, 
						q_xActive	=> xDetectOnlineChangeActive, 
						q_xReady	=> xDetectOnlineChangeReady, 
						q_etDiag	=> etDetectOnlineChangeDiag, 
						q_etDiagExt	=> etDetectOnlineChangeDiagExt, 
						q_sMsg		=> sDetectOnlineChangeMsg, 
						q_xChange	=> );
						
IF(NOT fbDetectOnlineChange.q_xChange) THEN
	RETURN;
END_IF

iq_stStandardModuleItf.iq_stExt.udiNumberOfSubModules 		:= c_udiNumberOfSubModules;
iq_stStandardModuleItf.iq_stExt.dwSubModulesItf		 		:= ADR(astSubModuleInterface);
iq_stStandardModuleItf.iq_stExt.pdwSubModulesAddItf		 	:= ADR(adwSubModuleAddInterfaces);
iq_stStandardModuleItf.iq_stExt.pstListofCMDTables			:= ADR(astListOfCMDTables);
iq_stStandardModuleItf.iq_stExt.udiNumberOfCmdTables		:= c_udiNumberOfCMDTables;
(* End of system generated code, do not change without consulting 'Schneider Electric Automation GmbH' - otherwise you risk instability!!!*)

(* System generated code, could be modified for your application *)
xUpdateStructsException := FALSE;

//-------------------------------------------------------------------------------------------------------------------
//-- Update CmdTable - Prepare 
	//
	TPL.FC_UpdateCmdTableListElement(	i_pstListofCmdTables	:= ADR(astListOfCmdTables),
										i_udiNumberOfCmdTables	:= c_udiNumberOfCmdTables,
										i_diCmd					:= ET_Cmd.Prepare,
										i_pstCmdTable			:= ADR(astPrepareTable),
										q_etDiag				=> etDiag,
										q_etDiagExt				=> etDiagExtTPL);
										
	IF etDiag <> GD.ET_Diag.Ok AND NOT xUpdateStructsException THEN
		xUpdateStructsException := TRUE;
		
		stUpdateStructsException.sMsg := PDL.FC_MultiConcat(i_sString1 := 'Update CmdTable: Prepare - ', 
															i_sString2 := GD.FC_EtDiagToString(i_etDiag := etDiag), 
															i_sString3 := ' - ', 
															i_sString4 := TPL.FC_EtDiagExtToString(i_etDiagExt := etDiagExtTPL));
	END_IF										

//-------------------------------------------------------------------------------------------------------------------
//-- Update CmdTable - Auto 
	//
	TPL.FC_UpdateCmdTableListElement(	i_pstListofCmdTables	:= ADR(astListOfCmdTables),
										i_udiNumberOfCmdTables	:= c_udiNumberOfCmdTables,
										i_diCmd					:= ET_Cmd.Auto,
										i_pstCmdTable			:= ADR(astAutoTable),
										q_etDiag				=> etDiag,
										q_etDiagExt				=> etDiagExtTPL);
										
	IF etDiag <> GD.ET_Diag.Ok AND NOT xUpdateStructsException THEN
		xUpdateStructsException := TRUE;
		
		stUpdateStructsException.sMsg := PDL.FC_MultiConcat(i_sString1 := 'Update CmdTable: Auto - ', 
															i_sString2 := GD.FC_EtDiagToString(i_etDiag := etDiag), 
															i_sString3 := ' - ', 
															i_sString4 := TPL.FC_EtDiagExtToString(i_etDiagExt := etDiagExtTPL));
	END_IF		

//-------------------------------------------------------------------------------------------------------------------
//-- Update CmdTable - Manual 
	//
	TPL.FC_UpdateCmdTableListElement(	i_pstListofCMDTables	:= ADR(astListofCMDTables),
										i_udiNumberOfCMDTables	:= c_udiNumberOfCMDTables,
										i_diCMD					:= ET_Cmd.Manual,
										i_pstCMDTable			:= ADR(astManualTable),
										q_etDiag				=> etDiag,
										q_etDiagExt				=> etDiagExtTPL);
										
	IF etDiag <> GD.ET_Diag.Ok AND NOT xUpdateStructsException THEN
		xUpdateStructsException := TRUE;
		
		stUpdateStructsException.sMsg := PDL.FC_MultiConcat(i_sString1 := 'Update CmdTable: Manual - ', 
															i_sString2 := GD.FC_EtDiagToString(i_etDiag := etDiag), 
															i_sString3 := ' - ', 
															i_sString4 := TPL.FC_EtDiagExtToString(i_etDiagExt := etDiagExtTPL));
	END_IF		

//-------------------------------------------------------------------------------------------------------------------
//-- Update CmdTable - Stop 
	//
	TPL.FC_UpdateCmdTableListElement(	i_pstListofCMDTables	:= ADR(astListofCMDTables),
										i_udiNumberOfCMDTables	:= c_udiNumberOfCMDTables,
										i_diCMD					:= ET_Cmd.Stop,
										i_pstCMDTable			:= ADR(astStopTable),
										q_etDiag				=> etDiag,
										q_etDiagExt				=> etDiagExtTPL);
										
	IF etDiag <> GD.ET_Diag.Ok AND NOT xUpdateStructsException THEN
		xUpdateStructsException := TRUE;
		
		stUpdateStructsException.sMsg := PDL.FC_MultiConcat(i_sString1 := 'Update CmdTable: Stop - ', 
															i_sString2 := GD.FC_EtDiagToString(i_etDiag := etDiag), 
															i_sString3 := ' - ', 
															i_sString4 := TPL.FC_EtDiagExtToString(i_etDiagExt := etDiagExtTPL));
	END_IF		

//-------------------------------------------------------------------------------------------------------------------
//-- Update CmdTable - Start 
	//
	TPL.FC_UpdateCmdTableListElement(	i_pstListofCMDTables	:= ADR(astListofCMDTables),
										i_udiNumberOfCmdTables	:= c_udiNumberOfCMDTables,
										i_diCMD					:= ET_Cmd.Start,
										i_pstCMDTable			:= ADR(astStartTable),
										q_etDiag				=> etDiag,
										q_etDiagExt				=> etDiagExtTPL);
										
	IF etDiag <> GD.ET_Diag.Ok AND NOT xUpdateStructsException THEN
		xUpdateStructsException := TRUE;
		
		stUpdateStructsException.sMsg := PDL.FC_MultiConcat(i_sString1 := 'Update CmdTable: Start - ', 
															i_sString2 := GD.FC_EtDiagToString(i_etDiag := etDiag), 
															i_sString3 := ' - ', 
															i_sString4 := TPL.FC_EtDiagExtToString(i_etDiagExt := etDiagExtTPL));
	END_IF		

//-------------------------------------------------------------------------------------------------------------------
//-- Update CmdTable - Abort 
	//
	TPL.FC_UpdateCmdTableListElement(	i_pstListofCMDTables	:= ADR(astListofCMDTables),
										i_udiNumberOfCmdTables	:= c_udiNumberOfCmdTables,
										i_diCMD					:= ET_Cmd.Abort,
										i_pstCMDTable			:= ADR(astAbortTable),
										q_etDiag				=> etDiag,
										q_etDiagExt				=> etDiagExtTPL);
										
	IF etDiag <> GD.ET_Diag.Ok AND NOT xUpdateStructsException THEN
		xUpdateStructsException := TRUE;
		
		stUpdateStructsException.sMsg := PDL.FC_MultiConcat(i_sString1 := 'Update CmdTable: Abort - ', 
															i_sString2 := GD.FC_EtDiagToString(i_etDiag := etDiag), 
															i_sString3 := ' - ', 
															i_sString4 := TPL.FC_EtDiagExtToString(i_etDiagExt := etDiagExtTPL));
	END_IF		

//-------------------------------------------------------------------------------------------------------------------
//-- Update CmdTable - Hold 
	//
	TPL.FC_UpdateCmdTableListElement(	i_pstListofCMDTables	:= ADR(astListofCMDTables),
										i_udiNumberOfCmdTables	:= c_udiNumberOfCmdTables,
										i_diCMD					:= ET_Cmd.Hold,
										i_pstCMDTable			:= ADR(astHoldTable),
										q_etDiag				=> etDiag,
										q_etDiagExt				=> etDiagExtTPL);
										
	IF etDiag <> GD.ET_Diag.Ok AND NOT xUpdateStructsException THEN
		xUpdateStructsException := TRUE;
		
		stUpdateStructsException.sMsg := PDL.FC_MultiConcat(i_sString1 := 'Update CmdTable: Hold - ', 
															i_sString2 := GD.FC_EtDiagToString(i_etDiag := etDiag), 
															i_sString3 := ' - ', 
															i_sString4 := TPL.FC_EtDiagExtToString(i_etDiagExt := etDiagExtTPL));
	END_IF		
				
//-------------------------------------------------------------------------------------------------------------------
//-- Update CmdTable - TestMulticarrier 
	//
	TPL.FC_UpdateCmdTableListElement(	i_pstListofCMDTables	:= ADR(astListofCMDTables),
										i_udiNumberOfCMDTables	:= c_udiNumberOfCMDTables,
										i_diCMD					:= ET_Cmd.TestMulticarrier,
										i_pstCMDTable			:= ADR(astTestMulticarrierTable),
										q_etDiag				=> etDiag,
										q_etDiagExt				=> etDiagExtTPL);
										
	IF etDiag <> GD.ET_Diag.Ok AND NOT xUpdateStructsException THEN
		xUpdateStructsException := TRUE;
		
		stUpdateStructsException.sMsg := PDL.FC_MultiConcat(i_sString1 := 'Update CmdTable: TestMulticarrier - ', 
															i_sString2 := GD.FC_EtDiagToString(i_etDiag := etDiag), 
															i_sString3 := ' - ', 
															i_sString4 := TPL.FC_EtDiagExtToString(i_etDiagExt := etDiagExtTPL));
	END_IF		
									
//-------------------------------------------------------------------------------------------------------------------
//-- Update CmdTable - TrackCalibration 
	//
	TPL.FC_UpdateCmdTableListElement(	i_pstListofCMDTables	:= ADR(astListofCMDTables),
										i_udiNumberOfCMDTables	:= c_udiNumberOfCMDTables,
										i_diCMD					:= ET_Cmd.TrackCalibration,
										i_pstCMDTable			:= ADR(astTrackCalibrationTable),
										q_etDiag				=> etDiag,
										q_etDiagExt				=> etDiagExtTPL);
										
	IF etDiag <> GD.ET_Diag.Ok AND NOT xUpdateStructsException THEN
		xUpdateStructsException := TRUE;
		
		stUpdateStructsException.sMsg := PDL.FC_MultiConcat(i_sString1 := 'Update CmdTable: TrackCalibration - ', 
															i_sString2 := GD.FC_EtDiagToString(i_etDiag := etDiag), 
															i_sString3 := ' - ', 
															i_sString4 := TPL.FC_EtDiagExtToString(i_etDiagExt := etDiagExtTPL));
	END_IF
//-------------------------------------------------------------------------------------------------------------------
//-- Update AddInterface - MultiCarrierTrack *)
	//	
	//AXM.FC_UpdateAddInterfaceStruct(	i_pdwSubModuleAddInterfaces	:= ADR(adwSubModuleAddInterfaces),
	//									i_udiSubModuleConstant		:= c_udiMultiCarrierTrack,
	//									iq_stAxisModuleItf			:= stMultiCarrierTrackInterface,
	//									q_etDiag					=> etDiag,
	//									q_etDiagExt					=> etDiagExtAXM);
	//									
	//IF etDiag <> GD.ET_Diag.Ok AND NOT xUpdateStructsException THEN
	//	xUpdateStructsException := TRUE;
	//	
	//	stUpdateStructsException.sMsg := PDL.FC_MultiConcat(i_sString1 := 'Update AddInterface: MultiCarrierTrack - ', 
	//														i_sString2 := GD.FC_EtDiagToString(i_etDiag := etDiag), 
	//														i_sString3 := ' - ', 
	//														i_sString4 := AXM.FC_EtDiagExtToString(i_etDiagExt := etDiagExtAXM));
	//END_IF		
	
//-------------------------------------------------------------------------------------------------------------------
//-- Set exception if any exception occurred *)
	//	
	fbExceptionHandler.SetException(i_xExceptionActive	:= xUpdateStructsException, 
									iq_stException		:= stUpdateStructsException, 
									iq_stExceptionList	:= iq_stExceptionList);
									
	xInitSuccessful := xInitSuccessful AND NOT xUpdateStructsException;
	
	etDiag := GD.ET_Diag.Ok;
//	

(* End of system generated code, could be modified for your application *)
END_ACTION

ACTION TrackCalibration_Logic:
IF xStartCalibration
AND xActiveFbTrackCalibration
AND xReadyFbTrackCalibration
THEN
	xStartCalibration := FALSE;
	
	fbTrackCalibration.StartCalibration(i_etMode		:= etModeTrackCalibration,
										q_xError		=> xSetException, 
										q_etResult		=> etResultMCR, 
										q_sResultMsg	=> sResultMsgMCR);
END_IF

IF xStartMeasurement
AND xActiveFbTrackCalibration
AND xReadyFbTrackCalibration
THEN
	xStartMeasurement := FALSE;
	
	fbTrackCalibration.StartMeasurement(i_etMode		:= etModeTrackCalibration,
										q_xError		=> xSetException, 
										q_etResult		=> etResultMCR, 
										q_sResultMsg	=> sResultMsgMCR);
END_IF


IF xResetTrackCalibration
AND xActiveFbTrackCalibration
AND xReadyFbTrackCalibration
THEN
	xResetTrackCalibration := FALSE;
	
	fbTrackCalibration.ResetTrackCalibration(	q_xError		=> xSetException, 
												q_etResult		=> etResultMCR, 
												q_sResultMsg	=> sResultMsgMCR);
END_IF
END_ACTION

END_PROGRAM

// LMC_PacDrive/Application/TemplateFullProgrammingFramework/EquipmentModules/MulticarrierModule/Multicarrier Stations/AutomaticMode/FB_Station1

FUNCTION_BLOCK FB_Station1 EXTENDS FB_MotionStationBase 
VAR
	
END_VAR

METHOD CyclicMotionCall : BOOL
VAR_IN_OUT
	iq_xTrigger : BOOL;
END_VAR
CASE iState OF

//----------------------------------------------------------------------------------------------------------------------------------- 
0: 	//--- Wait for Carrier in Station
	IF  THIS^.udiNumberOfCarriersInStationTotal > 0 
    THEN
				
		AddMessageToAPL('Move Carrier in Station '); 
													
		//--- get carrier -----------------------	
		GetStationCarrier(i_udiElementNumber := 1);
		
		//--- MoveGap -----------------------	
			MoveGap(
				i_etPosMode			:= MCR.ET_PosMode.AbsoluteForward, 
				i_lrTargetGap		:= THIS^.lrProcessGap, 
				i_lrTarget			:= THIS^.lrProcessPosition);
			
		IF NOT THIS^.xError_loc THEN
			iState := 10;
		END_IF
	END_IF

//----------------------------------------------------------------------------------------------------------------------------------- 
10: //--- Set Ready for next job 	
	IF THIS^.ifCarrier.ifFeedback.ifFeedbackMoveGapControl.xInEndTargetPosition  
	THEN
		THIS^.xStationReadyForJob_loc := TRUE; 
		iState := 20;
	END_IF
//----------------------------------------------------------------------------------------------------------------------------------- 
20: //--- Move Carrier Out of Station
	IF 	iq_xTrigger  THEN
		
		iq_xTrigger := FALSE;
 		
		AddMessageToAPL('Move Carrier out of Station '); 
		
		//--- write new MotionParameter  -----------------------	
			WriteMotionParameter(
				i_lrMaxVelocity     := THIS^.lrMaxVelocity,     
				i_lrMaxAcceleration := THIS^.lrMaxAcceleration, 
				i_lrMaxDeceleration := THIS^.lrMaxDeceleration, 
				i_lrMaxAbsJerk		:= THIS^.lrMaxJerk);      
       
		//--- MoveGap --------------------------------------------	
			MoveGap(
				i_etPosMode			:= MCR.ET_PosMode.AbsoluteForward, 
				i_lrTargetGap		:= THIS^.ifTargetStation.lrHandoverTargetGap, 
				i_lrTarget			:= THIS^.ifTargetStation.lrHandoverTargetPosition);
			
		//--- handover --------------------------------------------	
			HandoverCarriers(i_udiNumberOfCarriers := 1);
			
		//--- state jump ------------------------------------------	
			IF NOT THIS^.xError_loc THEN
				THIS^.xStationReadyForJob_loc := FALSE;
				iState := 0;
			END_IF
	END_IF
//----------------------------------------------------------------------------------------------------------------------------------- 

END_CASE
END_METHOD

END_FUNCTION_BLOCK

// LMC_PacDrive/Application/TemplateFullProgrammingFramework/EquipmentModules/MulticarrierModule/Multicarrier Stations/Test Multicarrier/SR_CallTestStations
PROGRAM SR_CallTestStations
VAR_INPUT
	i_etTraceSource  : ET_TraceSource;
	i_ifMultiCarrier : MCR.IF_Multicarrier;
	i_xStart	 	 : BOOL;
	i_xStop	 		 : BOOL;
END_VAR

VAR_OUTPUT
	q_xError	: BOOL;
	q_sEtResult 	: STRING(255);
	q_sResultMsg 	: STRING(255);
END_VAR


VAR
	
	uiSetOpModeVis					: UINT;
	uiSetOpModeTestVis				: UINT;
	uiStoredOpModeTestVis			: UINT := 999;

	udiLoop							: UDINT;
	etResultMCR						: MCR.ET_Result;
	fbLoggerPoint					: APL.FB_LoggerPoint;
	
	stZeroProductOffset				: MCR.PDL.ST_Vector3D;
	stZeroToolOffset				: MCR.PDL.ST_Vector3D;
END_VAR

//-- detect example change from vis
	IF uiSetOpModeTestVis <> uiStoredOpModeTestVis THEN
		
	//-- deactivate last example
		DeactivateLastTestStation();
		
	//-- activate new example
		ActivateSelectedTestStation();
		
		uiStoredOpModeTestVis := uiSetOpModeTestVis;

	END_IF
		
	//-- call selected example
	IF uiSetOpModeTestVis = 0 THEN
		SR_PlayGround(
			i_etTraceSource		:= i_etTraceSource,
			i_ifMultiCarrier	:= i_ifMultiCarrier,
			i_xStart			:= i_xStart,
			i_xStop				:= i_xStop,
			q_xError			=> q_xError,
			q_sEtResult			=> q_sEtResult,
			q_sResultMsg		=> q_sResultMsg);
			
	ELSIF uiSetOpModeTestVis = 1 THEN
		SR_SimpleStation(
			i_etTraceSource		:= i_etTraceSource,
			i_ifMultiCarrier	:= i_ifMultiCarrier,
			i_xStart			:= i_xStart,
			i_xStop				:= i_xStop,
			q_xError			=> q_xError,
			q_sEtResult			=> q_sEtResult,
			q_sResultMsg		=> q_sResultMsg);
			
	ELSIF uiSetOpModeTestVis = 2 THEN
		SR_PosAndSync(		
			i_etTraceSource		:= i_etTraceSource,
			i_ifMultiCarrier	:= i_ifMultiCarrier,
			i_xStart			:= i_xStart,
			i_xStop				:= i_xStop,
			q_xError			=> q_xError,
			q_sEtResult			=> q_sEtResult,
			q_sResultMsg		=> q_sResultMsg);
			
	ELSIF uiSetOpModeTestVis = 3 THEN
		SR_ColorStation(		
			i_etTraceSource		:= i_etTraceSource,
			i_ifMultiCarrier	:= i_ifMultiCarrier,
			i_xStart			:= i_xStart,
			i_xStop				:= i_xStop,
			q_xError			=> q_xError,
			q_sEtResult			=> q_sEtResult,
			q_sResultMsg		=> q_sResultMsg);
			
	ELSIF uiSetOpModeTestVis = 4 THEN
		SR_VelLimitStations(		
			i_etTraceSource		:= i_etTraceSource,
			i_ifMultiCarrier	:= i_ifMultiCarrier,
			i_xStart			:= i_xStart,
			i_xStop				:= i_xStop,
			q_xError			=> q_xError,
			q_sEtResult			=> q_sEtResult,
			q_sResultMsg		=> q_sResultMsg);
			
	ELSIF uiSetOpModeTestVis = 5 THEN
		SR_ClampingDeclamping(		
			i_etTraceSource		:= i_etTraceSource,
			i_ifMultiCarrier	:= i_ifMultiCarrier,
			i_xStart			:= i_xStart,
			i_xStop				:= i_xStop,
			q_xError			=> q_xError,
			q_sEtResult			=> q_sEtResult,
			q_sResultMsg		=> q_sResultMsg);
			
	ELSIF uiSetOpModeTestVis = 6 THEN
		SR_Grouping(		
			i_etTraceSource		:= i_etTraceSource,
			i_ifMultiCarrier	:= i_ifMultiCarrier,
			i_xStart			:= i_xStart,
			i_xStop				:= i_xStop,
			q_xError			=> q_xError,
			q_sEtResult			=> q_sEtResult,
			q_sResultMsg		=> q_sResultMsg);
			
	ELSIF uiSetOpModeTestVis = 7 THEN
		SR_ExternalMaster(		
			i_etTraceSource		:= i_etTraceSource,
			i_ifMultiCarrier	:= i_ifMultiCarrier,
			i_xStart			:= i_xStart,
			i_xStop				:= i_xStop,
			q_xError			=> q_xError,
			q_sEtResult			=> q_sEtResult,
			q_sResultMsg		=> q_sResultMsg);
			
	ELSIF uiSetOpModeTestVis = 8 THEN
		SR_Superimpose(		
			i_etTraceSource		:= i_etTraceSource,
			i_ifMultiCarrier	:= i_ifMultiCarrier,
			i_xStart			:= i_xStart,
			i_xStop				:= i_xStop,
			q_xError			=> q_xError,
			q_sEtResult			=> q_sEtResult,
			q_sResultMsg		=> q_sResultMsg);	
	END_IF

END_PROGRAM

// LMC_PacDrive/Application/TemplateFullProgrammingFramework/EquipmentModules/MulticarrierModule/SR_CarriersInStationToTrace
PROGRAM SR_CarriersInStationToTrace
VAR CONSTANT
	c_udiMaxNumberOfCarrierInTrace : UDINT := 5;
END_VAR

VAR
	fbDummyFeedback			:	MCR.FB_DummyCarrierFeedback;
	fbtrigger 				: Standard.R_Trig;
	raudiCarrierIndexArray	: REFERENCE TO ARRAY [1..MCR.GPl.Gc_udiMaxNumberOfCarriers] OF UDINT;
	udiLoop					: UDINT;
	udiTraceChannel			: UDINT;
END_VAR

VAR_INPUT
	i_xOneByOne		 	: BOOL;
	i_udiNumberOfCarrierInTrace : UDINT;
	i_ifMultiCarrier 	: MCR.IF_Multicarrier;
END_VAR

VAR_IN_OUT
	iq_xReStartSerialCount: BOOL;
END_VAR

VAR_OUTPUT
	q_aifTraceObject	: ARRAY[1..c_udiMaxNumberOfCarrierInTrace] OF MCR.IF_CarrierFeedback  := [c_udiMaxNumberOfCarrierInTrace(fbDummyFeedback)];;
END_VAR

METHOD Call
VAR_INPUT
	i_xTrigger : BOOL;
	i_ifStation	: MCRS.IF_CoreStation;
END_VAR
fbtrigger(CLK := i_xTrigger);

//--- parallel ----
IF 		fbtrigger.Q
	AND_THEN i_ifStation <> 0
	AND_THEN i_ifStation.udiNumberOfCarriersInStationTotal > 0
	AND_THEN NOT i_xOneByOne
THEN
	raudiCarrierIndexArray REF= i_ifStation.raudiCarrierIndexArray;
	
	FOR udiLoop := 1 TO MIN(i_ifStation.udiNumberOfCarriersInStationTotal,MIN(i_udiNumberOfCarrierInTrace,c_udiMaxNumberOfCarrierInTrace)) DO
		q_aifTraceObject[udiLoop] := i_ifMultiCarrier.raifCarrier[raudiCarrierIndexArray[udiLoop]].ifFeedback;
	END_FOR
	
END_IF

//--- serial ----
IF 		fbtrigger.Q
	AND_THEN i_ifStation <> 0
	AND_THEN i_ifStation.udiNumberOfCarriersInStationTotal > 0
	AND_THEN i_xOneByOne
THEN	
	raudiCarrierIndexArray REF= i_ifStation.raudiCarrierIndexArray;
	
	udiTraceChannel := udiTraceChannel + 1; 
	
	IF 			udiTraceChannel > MIN(i_udiNumberOfCarrierInTrace,c_udiMaxNumberOfCarrierInTrace) 
		OR_ELSE iq_xReStartSerialCount 
	THEN
		iq_xReStartSerialCount := FALSE;
		udiTraceChannel := 1; 
	END_IF 
	
	q_aifTraceObject[udiTraceChannel] := i_ifMultiCarrier.raifCarrier[raudiCarrierIndexArray[1]].ifFeedback;
END_IF
END_METHOD

END_PROGRAM

// LMC_PacDrive/Application/TemplateFullProgrammingFramework/EquipmentModules/MulticarrierModule/FC_SplitString
FUNCTION FC_SplitString : BOOL
VAR_INPUT
	i_sString	: STRING(255);
END_VAR
VAR_OUTPUT
	q_sString1	: STRING(80);
	q_sString2	: STRING(80);
	q_sString3	: STRING(80);
END_VAR

VAR
	iPositionSpace	: INT;
	sRestString		: STRING(255);
	iHalfLen		: INT;
	iRepeatCounter   : INT; //Counter for interrupt Repeat-loop to avoid deadlock
END_VAR

VAR_STAT
	sLastString : STRING(255);
	sString1	: STRING(80);
	sString2	: STRING(80);
	sString3	: STRING(80);
END_VAR

IF sLastString <> i_sString THEN //--- split string only once
	sLastString := i_sString;
	sString1 := '';
	sString2 := '';
	sString3 := '';
	
	//--- string is less than 70 characters
	IF Standard.LEN(i_sString) < 70 THEN
		sString1 := i_sString;
		RETURN;
	END_IF
	
	//--- split first part
	iHalfLen := Standard.LEN(i_sString) / 2;
	
	sRestString := i_sString;
	sString1	:= Left(sRestString,find(sRestString,' '));
	// split string
	REPEAT
		iRepeatCounter := iRepeatCounter + 1;
		
		IF LEN(sString1) < 70 OR LEN(sString1) < iHalfLen THEN
			sRestString 	:= Standard.DELETE(sRestString,find(sRestString,' '),1);  
			sString1		:= Standard.CONCAT(sString1,(Left(sRestString,find(sRestString,' '))));
		END_IF 
		
	UNTIL LEN(sString1) >= 70 OR LEN(sString1) >= iHalfLen OR iRepeatCounter > 20
	END_REPEAT
		
	sRestString 	:= Standard.DELETE(sRestString,find(sRestString,' '),1);  
	sString2 		:= sRestString;
	
	//--- check if second split is necessary
	IF Standard.LEN(sRestString) < 70 THEN
		RETURN;
	END_IF
	
	//--- split second part
	iRepeatCounter 	:= 0;
	iHalfLen 		:= Standard.LEN(sRestString) / 2;
	sString2		:= Left(sRestString,find(sRestString,' '));
	REPEAT
		iRepeatCounter := iRepeatCounter + 1;
		
		IF LEN(sString2) < 70 OR LEN(sString2) < iHalfLen THEN
			sRestString 	:= Standard.DELETE(sRestString,find(sRestString,' '),1);  
			sString2		:= Standard.CONCAT(sString2,(Left(sRestString,find(sRestString,' '))));
		END_IF 
		
	UNTIL LEN(sString2) >= 70 OR LEN(sString2) >= iHalfLen OR iRepeatCounter > 20
	END_REPEAT
	
	sRestString 	:= Standard.DELETE(sRestString,find(sRestString,' '),1);  
	sString3 		:= sRestString;
	
ELSE
	q_sString1 		:= sString1;
	q_sString2 		:= sString2;
	q_sString3 		:= sString3;
END_IF

END_FUNCTION

// LMC_PacDrive/Application/TemplateFullProgrammingFramework/Tools/FC_ObjectTypeIsMotionAxis
(* Checks whether the given diObjectType is an object representing a Motion Axis (drive beneath Sercos_Master bus) *)
FUNCTION FC_ObjectTypeIsMotionAxis : BOOL

VAR_INPUT
	i_udiObjectType: UDINT; (* Type (UDINT) of object to be checked to be a motion axis *)  
END_VAR

(* Currently, this implemetation is hacky. We compare the ObjectType to a static list of ObjectTypes known as Motion Drives.
   What we acutlly want is to get the IEC object by LogicalAddress and check whether it fits the interface IF_Drive. But sadly, 
   such a function doesn't exist yet *)

IF	i_udiObjectType = SystemInterface.LXM62DxS_TYPE.udiType OR_ELSE
	i_udiObjectType = SystemInterface.ILM62_TYPE.udiType OR_ELSE
	i_udiObjectType = SystemInterface.LXM52_TYPE.udiType OR_ELSE
	i_udiObjectType = SystemInterface.SERCDRV_TYPE.udiType OR_ELSE
	i_udiObjectType = SystemInterface.LXM52Linear_TYPE.udiType OR_ELSE
	i_udiObjectType = SystemInterface.LXM62DxSLinear_TYPE.udiType OR_ELSE
	i_udiObjectType = SystemInterface.LXMMCC_TYPE.udiType OR_ELSE 
	i_udiObjectType = SystemInterface.LXMMCS_TYPE.udiType  
	
THEN
   FC_ObjectTypeIsMotionAxis := TRUE;
ELSE
   FC_ObjectTypeIsMotionAxis := FALSE;
END_IF

RETURN;

END_FUNCTION

// LMC_PacDrive/Application/TemplateFullProgrammingFramework/TaskCalls/SR_ReadControlLoopParameter
PROGRAM SR_ReadControlLoopParameter

VAR_OUTPUT
	q_xReadParameterDone				: BOOL;
	q_xReadParameterError				: BOOL;
END_VAR


VAR
	dwPosP_Straight				: DWORD;
	dwVelP_Straight				: DWORD;
	dwVelI_Straight				: DWORD; 
	
	dwPosP_Curve				: DWORD;
	dwVelP_Curve				: DWORD;
	dwVelI_Curve				: DWORD; 

	xStart						: BOOL;
	diState						: DINT;
	
	//-- Sercos IDNs
	dwIDNCarrierPosP					: DWORD := SERC.FC_BuildIDN(0, 18, TRUE,  0, 1089); //P-0-1089.0.18 
	dwIDNCarrierVelP					: DWORD := SERC.FC_BuildIDN(0, 15, TRUE,  0, 1089); //P-0-1089.0.15
	dwIDNCarrierVelI					: DWORD := SERC.FC_BuildIDN(0, 16, TRUE,  0, 1089); //P-0-1089.0.16  
	
 	dwIDNCarrierMaxcurr               	: DWORD := SERC.FC_BuildIDN(0, 0,  TRUE,  0, 0208); //P-0-0208.0.0  
    dwIDNCarrierLoad                  	: DWORD := SERC.FC_BuildIDN(0, 14, TRUE,  0, 1089); //P-0-1089.0.14,    
    dwIDNDeviationLevelWarning        	: DWORD := SERC.FC_BuildIDN(0, 0,  TRUE,  0, 2014); //P-0-2014.0.0 Warning
    dwIDNDeviationLevelError          	: DWORD := SERC.FC_BuildIDN(0, 1,  TRUE,  0, 2014); //P-0-2014.0.1 Error

	diResultSercosReadServiceData	  	: DINT;	

	dwMaxCurr			              	: DWORD;
    dwMaxload					      	: DWORD;
    dwDeviationLevelWarning           	: DWORD;
    dwDeviationLevelError             	: DWORD; 

	uiReadDataLen						: UINT;
	uiMaxReadDataLen					: UINT;
	udiIndex							: UDINT;
	udiStraightIndex					: UDINT;
	udiCurveIndex						: UDINT;
END_VAR

CASE diState OF
	
	//-------------------------------------------------------------------------------------------------------------------------------------------
	0:	//--- Wait for start
		
		IF xStart THEN
			xStart	:= FALSE;
			udiStraightIndex := 0;
			udiCurveIndex	 := 0;
			//-- Get straight segment
			FOR udiIndex := 1  TO GVL_MulticarrierConfiguration.Gc_astTracks[1].udiNumberOfSegments DO
				IF NOT GVL_MulticarrierConfiguration.Gc_astSegmentTypes[GVL_MulticarrierConfiguration.Gc_astTracks[1].astSegments[udiIndex].diSegmentTypesIndex].xIsCurved  
				THEN
					udiStraightIndex	 := udiIndex;
					EXIT;
				END_IF
			END_FOR  
			
			//-- Get curve segment
			FOR udiIndex := 1  TO GVL_MulticarrierConfiguration.Gc_astTracks[1].udiNumberOfSegments DO
				IF GVL_MulticarrierConfiguration.Gc_astSegmentTypes[GVL_MulticarrierConfiguration.Gc_astTracks[1].astSegments[udiIndex].diSegmentTypesIndex].xIsCurved  
				THEN
					udiCurveIndex	  := udiIndex;
					EXIT;
				END_IF
			END_FOR  
			diState := 10;
		END_IF
		
	//-------------------------------------------------------------------------------------------------------------------------------------------
	10:	//--- ReadParameter: Pos_P AllSegments
		uiReadDataLen	 := 4;
		uiMaxReadDataLen := 4;
		diResultSercosReadServiceData 	:= SercosReadServiceDataFromSegments(	i_dwIDN					:= dwIDNCarrierPosP, 
																				i_udiStraightIndex      := udiStraightIndex,
																				q_dwDataStraightSegment	=> dwPosP_Straight, 
																				i_udiCurveIndex		    := udiCurveIndex,
																				q_dwDataCurveSegment	=> dwPosP_Curve,
																				i_wMaxDataLength		:= 4,
																				iq_uiReadDataLen		:= uiReadDataLen,
																				iq_uiMaxReadDataLen		:= uiMaxReadDataLen);
		IF diResultSercosReadServiceData = 0 THEN
			diState := 20;
		ELSE
			q_xReadParameterError	:= TRUE;
			diState	:= 1000;
		END_IF
		
	//-------------------------------------------------------------------------------------------------------------------------------------------
	20:	//--- ReadParameter Vel_P AllSegments
		uiReadDataLen	 := 4;
		uiMaxReadDataLen := 4;
		diResultSercosReadServiceData 	:= SercosReadServiceDataFromSegments(	i_dwIDN					:= dwIDNCarrierVelP, 
																				i_udiStraightIndex      := udiStraightIndex,
																				q_dwDataStraightSegment	=> dwVelP_Straight, 
																				i_udiCurveIndex		    := udiCurveIndex,
																				q_dwDataCurveSegment	=> dwVelP_Curve,
																				i_wMaxDataLength		:= 4,
																				iq_uiReadDataLen		:= uiReadDataLen,
																				iq_uiMaxReadDataLen		:= uiMaxReadDataLen);		
		IF diResultSercosReadServiceData = 0 THEN
			diState := 30;
		ELSE
			q_xReadParameterError	:= TRUE;
			diState	:= 1000;
		END_IF
	
	//-------------------------------------------------------------------------------------------------------------------------------------------
	30:	//--- ReadParameter Vel_I AllSegments
		uiReadDataLen	 := 4;
		uiMaxReadDataLen := 4;
		diResultSercosReadServiceData 	:= SercosReadServiceDataFromSegments(	i_dwIDN					:= dwIDNCarrierVelI, 
																				i_udiStraightIndex      := udiStraightIndex,
																				q_dwDataStraightSegment	=> dwVelI_Straight, 
																				i_udiCurveIndex		    := udiCurveIndex,
																				q_dwDataCurveSegment	=> dwVelI_Curve,
																				i_wMaxDataLength		:= 4,
																				iq_uiReadDataLen		:= uiReadDataLen,
																				iq_uiMaxReadDataLen		:= uiMaxReadDataLen);		
		IF diResultSercosReadServiceData = 0 THEN
			diState	:= 40;
		ELSE
			q_xReadParameterError	:= TRUE;
			diState	:= 1000;
		END_IF	
		
	//-------------------------------------------------------------------------------------------------------------------------------------------
	40: //--- ReadParameter TrackingDeviation WarningLevel AllSegments
		uiReadDataLen	 := 4;
		uiMaxReadDataLen := 4;
		diResultSercosReadServiceData := SercosReadServiceDataFromSegments( 	i_dwIDN 				:= dwIDNDeviationLevelWarning,
																				i_udiStraightIndex      := udiStraightIndex,
																				q_dwDataStraightSegment	=> dwDeviationLevelWarning,
																				i_udiCurveIndex		    := udiCurveIndex,
																				q_dwDataCurveSegment	=> dwDeviationLevelWarning,
																				i_wMaxDataLength 		:= 4,
																				iq_uiReadDataLen		:= uiReadDataLen,
																				iq_uiMaxReadDataLen		:= uiMaxReadDataLen);		
		IF diResultSercosReadServiceData = 0 THEN
			diState := 50;
		ELSE
			q_xReadParameterError	:= TRUE;
			diState := 1000;
		END_IF

	//-------------------------------------------------------------------------------------------------------------------------------------------
	50: //--- ReadParameter TrackingDeviation ErrorLevel AllSegments
		uiReadDataLen	 := 4;
		uiMaxReadDataLen := 4;
		diResultSercosReadServiceData := SercosReadServiceDataFromSegments( 	i_dwIDN 				:= dwIDNDeviationLevelError,
																				i_udiStraightIndex      := udiStraightIndex,
																				q_dwDataStraightSegment	=> dwDeviationLevelError,
																				i_udiCurveIndex		    := udiCurveIndex,
																				q_dwDataCurveSegment	=> dwDeviationLevelError,
																				i_wMaxDataLength 		:= 4,
																				iq_uiReadDataLen		:= uiReadDataLen,
																				iq_uiMaxReadDataLen		:= uiMaxReadDataLen);		
		IF diResultSercosReadServiceData = 0 THEN
			diState := 60;
		ELSE
			q_xReadParameterError	:= TRUE;
			diState := 1000;
		END_IF		
		
	//-------------------------------------------------------------------------------------------------------------------------------------------
	60:	//--- ReadParameter: Maximum Current AllSegments
	
		uiReadDataLen	 := 2;
		uiMaxReadDataLen := 2;
		diResultSercosReadServiceData 	:= SercosReadServiceDataFromSegments(	i_dwIDN					:= dwIDNCarrierMaxcurr, 
																				i_udiStraightIndex      := udiStraightIndex,
																				q_dwDataStraightSegment	=> dwMaxCurr, 
																				i_udiCurveIndex		    := udiCurveIndex,
																				q_dwDataCurveSegment	=> dwMaxCurr,
																				i_wMaxDataLength		:= 2,
																				iq_uiReadDataLen		:= uiReadDataLen,
																				iq_uiMaxReadDataLen		:= uiMaxReadDataLen);		
		IF diResultSercosReadServiceData = 0 THEN
			diState := 70;
		ELSE
			q_xReadParameterError	:= TRUE;
			diState	:= 1000;
		END_IF	
	
	//-------------------------------------------------------------------------------------------------------------------------------------------
	70:	//--- ReadParameter: Load of Carrier AllSegments
		uiReadDataLen	 := 4;
		uiMaxReadDataLen := 4;
		diResultSercosReadServiceData 	:= SercosReadServiceDataFromSegments(	i_dwIDN					:= dwIDNCarrierLoad, 
																				i_udiStraightIndex      := udiStraightIndex,
																				q_dwDataStraightSegment	=> dwMaxload, 
																				i_udiCurveIndex		    := udiCurveIndex,
																				q_dwDataCurveSegment	=> dwMaxload, 
																				i_wMaxDataLength		:= 4,
																				iq_uiReadDataLen		:= uiReadDataLen,
																				iq_uiMaxReadDataLen		:= uiMaxReadDataLen);		
		IF diResultSercosReadServiceData = 0 THEN
			q_xReadParameterDone	:= TRUE;
			diState := 0;
		ELSE
			q_xReadParameterError	:= TRUE;
			diState	:= 1000;
		END_IF	
	
	//-------------------------------------------------------------------------------------------------------------------------------------------
	1000: //--- ErrorState
		;
	
END_CASE

METHOD GetParameter
VAR_OUTPUT
	q_dwPosP_Straight				: DWORD;
	q_dwVelP_Straight				: DWORD;
	q_dwVelI_Straight				: DWORD;  
	q_dwPosP_Curve					: DWORD;
	q_dwVelP_Curve					: DWORD;
	q_dwVelI_Curve					: DWORD;  
	q_dwMaxCurr			            : DWORD;
    q_dwMaxload					    : DWORD;
    q_dwDeviationLevelWarning       : DWORD;
    q_dwDeviationLevelError         : DWORD; 
END_VAR
IF q_xReadParameterDone THEN
	
	q_dwPosP_Straight	:= 	dwPosP_Straight;
	q_dwVelP_Straight	:=	dwVelP_Straight;
	q_dwVelI_Straight	:=	dwVelI_Straight;
	
	q_dwPosP_Curve	:= 	dwPosP_Curve;
	q_dwVelP_Curve	:=	dwVelP_Curve;
	q_dwVelI_Curve	:=	dwVelI_Curve;

	q_dwMaxCurr			            := dwMaxCurr;
    q_dwMaxload					    := dwMaxload;
    q_dwDeviationLevelWarning       := dwDeviationLevelWarning;
    q_dwDeviationLevelError         := dwDeviationLevelError; 
	
END_IF
END_METHOD

METHOD ReadParameter
xStart 		:=  TRUE;
END_METHOD

METHOD SercosReadServiceDataFromSegments : DINT
VAR_INPUT
	i_dwIDN					: DWORD;
	i_udiCurveIndex			: UDINT;	
	i_udiStraightIndex		: UDINT;
	i_wMaxDataLength		: WORD;
END_VAR
VAR_OUTPUT
	q_dwDataCurveSegment	: DWORD;	
	q_dwDataStraightSegment	: DWORD;	
	
END_VAR
VAR_IN_OUT
	iq_uiReadDataLen 	: UINT;
	iq_uiMaxReadDataLen : UINT;
END_VAR
VAR
	dwDataCurveSegment		: DWORD;
	dwDataStraightSegment	: DWORD;
END_VAR
//-- Read straight segment Parameter
IF  i_udiStraightIndex > 0 THEN        
        SercosReadServiceDataFromSegments := SystemInterface.FC_SercosReadServiceDataByTopAddr(    
                                                                    i_wTopoAddr         := TO_WORD(i_udiStraightIndex), 
                                                                    i_dwIDN             := i_dwIDN,
                                                                    i_wType             := 5,
                                                                    i_dwPointerToData   := ADR(dwDataStraightSegment),
                                                                    i_wMaxDataLen       := i_wMaxDataLength,
																	iq_uiReadDataLen	:= iq_uiReadDataLen, 
																	iq_uiMaxReadDataLen	:= iq_uiMaxReadDataLen);
		q_dwDataStraightSegment := dwDataStraightSegment;
END_IF

IF SercosReadServiceDataFromSegments <> 0 THEN
	RETURN;
END_IF

//-- Read curve segment Parameter
 IF  i_udiCurveIndex > 0 THEN        
       SercosReadServiceDataFromSegments := SystemInterface.FC_SercosReadServiceDataByTopAddr(    
                                                                    i_wTopoAddr         := TO_WORD(i_udiCurveIndex), 
                                                                    i_dwIDN             := i_dwIDN,
                                                                    i_wType             := 5,
                                                                    i_dwPointerToData   := ADR(dwDataCurveSegment),
                                                                    i_wMaxDataLen       := i_wMaxDataLength,
																	iq_uiReadDataLen	:= iq_uiReadDataLen, 
																	iq_uiMaxReadDataLen	:= iq_uiMaxReadDataLen);
		q_dwDataCurveSegment := dwDataCurveSegment;
END_IF
END_METHOD

END_PROGRAM

// LMC_PacDrive/Application/TemplateFullProgrammingFramework/TaskCalls/SR_WriteControlLoopParameter
PROGRAM SR_WriteControlLoopParameter

VAR_OUTPUT
	q_xWriteParameterDone				: BOOL;
	q_xWriteParameterError				: BOOL;
END_VAR


VAR
	dwPosP_Straight				: DWORD;
	dwVelP_Straight				: DWORD;
	dwVelI_Straight				: DWORD; 
	
	dwPosP_Curve				: DWORD;
	dwVelP_Curve				: DWORD;
	dwVelI_Curve				: DWORD; 

	xStart						: BOOL;
	diState						: DINT;
	
	//-- Sercos IDNs
	dwIDNCarrierPosP					: DWORD := SERC.FC_BuildIDN(0, 18, TRUE,  0, 1089); //P-0-1089.0.18 
	dwIDNCarrierVelP					: DWORD := SERC.FC_BuildIDN(0, 15, TRUE,  0, 1089); //P-0-1089.0.15
	dwIDNCarrierVelI					: DWORD := SERC.FC_BuildIDN(0, 16, TRUE,  0, 1089); //P-0-1089.0.16  
	
 	dwIDNCarrierMaxcurr               	: DWORD := SERC.FC_BuildIDN(0, 0,  TRUE,  0, 0208); //P-0-0208.0.0  
    dwIDNCarrierLoad                  	: DWORD := SERC.FC_BuildIDN(0, 14, TRUE,  0, 1089); //P-0-1089.0.14    
    dwIDNDeviationLevelWarning        	: DWORD := SERC.FC_BuildIDN(0, 0,  TRUE,  0, 2014); //P-0-2014.0.0 
    dwIDNDeviationLevelError          	: DWORD := SERC.FC_BuildIDN(0, 1,  TRUE,  0, 2014); //P-0-2014.0.1 

	diResultSercosWriteServiceData	  	: DINT;	

	dwMaxCurr			              	: DWORD;
    dwMaxload					      	: DWORD;
    dwDeviationLevelWarning           	: DWORD;
    dwDeviationLevelError             	: DWORD;

END_VAR

CASE diState OF
	
	//-------------------------------------------------------------------------------------------------------------------------------------------
	0:	//--- Wait for start
		
		IF xStart THEN
			xStart	:= FALSE;
			diState := 10;
		END_IF
		
	//-------------------------------------------------------------------------------------------------------------------------------------------
	10:	//--- WriteParameter: Pos_P AllSegments
		diResultSercosWriteServiceData 	:= SercosWriteServiceDataToAllSegments(	i_dwIDN					:= dwIDNCarrierPosP, 
																				i_dwDataStraightSegment	:= dwPosP_Straight, 
																				i_dwDataCurveSegment	:= dwPosP_Curve,
																				i_wMaxDataLength		:= 4);
		IF diResultSercosWriteServiceData = 0 THEN
			diState := 20;
		ELSE
			q_xWriteParameterError	:= TRUE;
			diState	:= 1000;
		END_IF
		
	//-------------------------------------------------------------------------------------------------------------------------------------------
	20:	//--- WriteParameter Vel_P AllSegments
		diResultSercosWriteServiceData 	:= SercosWriteServiceDataToAllSegments(	i_dwIDN					:= dwIDNCarrierVelP, 
																				i_dwDataStraightSegment	:= dwVelP_Straight, 
																				i_dwDataCurveSegment	:= dwVelP_Curve,
																				i_wMaxDataLength		:= 4);
		IF diResultSercosWriteServiceData = 0 THEN
			diState := 30;
		ELSE
			q_xWriteParameterError	:= TRUE;
			diState	:= 1000;
		END_IF
	
